LIN {X 0,Y 396.421,Z 620.372,A -85,B 0,C 180,E1 -11060.818,E2 -11060.818} C_VEL
LIN {X 0,Y 396.005,Z 626.08,A -85,B 0,C 180,E1 -11062.862,E2 -11062.862} C_VEL
LIN {X 0,Y 395.858,Z 630.229,A -85,B 0,C 180,E1 -11064.906,E2 -11064.906} C_VEL
LIN {X 0,Y 395.697,Z 632.948,A -85,B 0,C 180,E1 -11066.944,E2 -11066.944} C_VEL
LIN {X 0,Y 395.755,Z 634.313,A -85,B 0,C 180,E1 -11068.981,E2 -11068.981} C_VEL
LIN {X 0,Y 395.755,Z 634.351,A -85,B 0,C 180,E1 -11071.016,E2 -11071.016} C_VEL
LIN {X 0,Y 395.696,Z 633.059,A -85,B 0,C 180,E1 -11073.053,E2 -11073.053} C_VEL
LIN {X 0,Y 395.856,Z 630.406,A -85,B 0,C 180,E1 -11075.091,E2 -11075.091} C_VEL
LIN {X 0,Y 396.003,Z 626.321,A -85,B 0,C 180,E1 -11077.135,E2 -11077.135} C_VEL
LIN {X 0,Y 396.407,Z 620.682,A -85,B 0,C 180,E1 -11079.18,E2 -11079.18} C_VEL
LIN {X 0,Y 396.918,Z 614.321,A -85,B 0,C 180,E1 -11080.971,E2 -11080.971} C_VEL
LIN {X 0,Y 397.802,Z 606.411,A -85,B 0,C 180,E1 -11082.757,E2 -11082.757} C_VEL
LIN {X 0,Y 398.55,Z 598.138,A -85,B 0,C 180,E1 -11084.291,E2 -11084.291} C_VEL
LIN {X 0,Y 399.604,Z 588.172,A -85,B 0,C 180,E1 -11085.818,E2 -11085.818} C_VEL
LIN {X 0,Y 400.764,Z 577.081,A -85,B 0,C 180,E1 -11087.212,E2 -11087.212} C_VEL
LIN {X 0,Y 401.87,Z 566.044,A -85,B 0,C 180,E1 -11088.347,E2 -11088.347} C_VEL
LIN {X 0,Y 402.968,Z 554.065,A -85,B 0,C 180,E1 -11089.35,E2 -11089.35} C_VEL
LIN {X 0,Y 404.005,Z 540.311,A -85,B 0,C 180,E1 -11090.255,E2 -11090.255} C_VEL
LIN {X 0,Y 404.838,Z 526.291,A -85,B 0,C 180,E1 -11090.946,E2 -11090.946} C_VEL
LIN {X 0,Y 405.521,Z 512.757,A -85,B 0,C 180,E1 -11091.408,E2 -11091.408} C_VEL
LIN {X 0,Y 405.97,Z 492.817,A -85,B 0,C 180,E1 -11091.816,E2 -11091.816} C_VEL
LIN {X 0,Y 407.438,Z 401.297,A -85,B 0,C 180,E1 -11093.445,E2 -11093.445} C_VEL
LIN {X 0,Y 402.179,Z 375.662,A -85,B 0,C 180,E1 -11094.261,E2 -11094.261} C_VEL
LIN {X 0,Y 401.525,Z 372.237,A -85,B 0,C 180,E1 -11094.402,E2 -11094.402} C_VEL
LIN {X 0,Y 401.284,Z 368.64,A -85,B 0,C 180,E1 -11095.131,E2 -11095.131} C_VEL
LIN {X 0,Y 398.971,Z 357.321,A -85,B 0,C 180,E1 -11097.727,E2 -11097.727} C_VEL
LIN {X 0,Y 397.187,Z 349.822,A -85,B 0,C 180,E1 -11099.551,E2 -11099.551} C_VEL
LIN {X 0,Y 397.111,Z 349.638,A -85,B 0,C 180,E1 -11103.271,E2 -11103.271} C_VEL
LIN {X 0,Y 397.105,Z 349.636,A -85,B 0,C 180,E1 -11105.733,E2 -11105.733} C_VEL
LIN {X 0,Y 397.111,Z 349.632,A -85,B 0,C 180,E1 -11109.575,E2 -11109.575} C_VEL
LIN {X 0,Y 397.154,Z 349.64,A -85,B 0,C 180,E1 -11112.254,E2 -11112.254} C_VEL
LIN {X 0,Y 397.145,Z 349.618,A -85,B 0,C 180,E1 -11115.058,E2 -11115.058} C_VEL
LIN {X 0,Y 397.149,Z 349.642,A -85,B 0,C 180,E1 -11118.005,E2 -11118.005} C_VEL
LIN {X 0,Y 397.102,Z 349.617,A -85,B 0,C 180,E1 -11121.725,E2 -11121.725} C_VEL
LIN {X 0,Y 397.117,Z 349.642,A -85,B 0,C 180,E1 -11125.506,E2 -11125.506} C_VEL
LIN {X 0,Y 397.076,Z 349.628,A -85,B 0,C 180,E1 -11129.117,E2 -11129.117} C_VEL
LIN {X 0,Y 397.185,Z 349.612,A -85,B 0,C 180,E1 -11132.609,E2 -11132.609} C_VEL
LIN {X 0,Y 397.124,Z 349.642,A -85,B 0,C 180,E1 -11135.981,E2 -11135.981} C_VEL
LIN {X 0,Y 397.128,Z 349.636,A -85,B 0,C 180,E1 -11139.704,E2 -11139.704} C_VEL
LIN {X 0,Y 397.171,Z 349.634,A -85,B 0,C 180,E1 -11142.844,E2 -11142.844} C_VEL
LIN {X 0,Y 397.215,Z 349.626,A -85,B 0,C 180,E1 -11146.678,E2 -11146.678} C_VEL
LIN {X 0,Y 397.219,Z 349.615,A -85,B 0,C 180,E1 -11149.809,E2 -11149.809} C_VEL
LIN {X 0,Y 397.354,Z 349.611,A -85,B 0,C 180,E1 -11152.888,E2 -11152.888} C_VEL
LIN {X 0,Y 397.248,Z 349.625,A -85,B 0,C 180,E1 -11154.925,E2 -11154.925} C_VEL
LIN {X 0,Y 397.442,Z 349.595,A -85,B 0,C 180,E1 -11157.973,E2 -11157.973} C_VEL
LIN {X 0,Y 397.574,Z 349.584,A -85,B 0,C 180,E1 -11160,E2 -11160} C_VEL
LIN {X 0,Y 397.374,Z 349.599,A -85,B 0,C 180,E1 -11163.041,E2 -11163.041} C_VEL
LIN {X 0,Y 397.353,Z 349.611,A -85,B 0,C 180,E1 -11167.112,E2 -11167.112} C_VEL
LIN {X 0,Y 397.219,Z 349.615,A -85,B 0,C 180,E1 -11170.191,E2 -11170.191} C_VEL
LIN {X 0,Y 397.215,Z 349.625,A -85,B 0,C 180,E1 -11173.321,E2 -11173.321} C_VEL
LIN {X 0,Y 397.171,Z 349.633,A -85,B 0,C 180,E1 -11177.156,E2 -11177.156} C_VEL
LIN {X 0,Y 397.104,Z 349.634,A -85,B 0,C 180,E1 -11180.73,E2 -11180.73} C_VEL
LIN {X 0,Y 397.124,Z 349.641,A -85,B 0,C 180,E1 -11184.019,E2 -11184.019} C_VEL
LIN {X 0,Y 397.184,Z 349.612,A -85,B 0,C 180,E1 -11187.391,E2 -11187.391} C_VEL
LIN {X 0,Y 397.069,Z 349.628,A -85,B 0,C 180,E1 -11190.883,E2 -11190.883} C_VEL
LIN {X 0,Y 397.117,Z 349.642,A -85,B 0,C 180,E1 -11194.494,E2 -11194.494} C_VEL
LIN {X 0,Y 397.101,Z 349.616,A -85,B 0,C 180,E1 -11198.275,E2 -11198.275} C_VEL
LIN {X 0,Y 397.149,Z 349.642,A -85,B 0,C 180,E1 -11201.995,E2 -11201.995} C_VEL
LIN {X 0,Y 397.144,Z 349.618,A -85,B 0,C 180,E1 -11205.061,E2 -11205.061} C_VEL
LIN {X 0,Y 397.15,Z 349.641,A -85,B 0,C 180,E1 -11208.008,E2 -11208.008} C_VEL
LIN {X 0,Y 397.104,Z 349.643,A -85,B 0,C 180,E1 -11211.727,E2 -11211.727} C_VEL
LIN {X 0,Y 397.121,Z 349.643,A -85,B 0,C 180,E1 -11215.508,E2 -11215.508} C_VEL
LIN {X 0,Y 397.084,Z 349.641,A -85,B 0,C 180,E1 -11219.12,E2 -11219.12} C_VEL
LIN {X 0,Y 397.147,Z 349.731,A -85,B 0,C 180,E1 -11220.445,E2 -11220.445} C_VEL
LIN {X 0,Y 399.635,Z 360.386,A -85,B 0,C 180,E1 -11223.033,E2 -11223.033} C_VEL
LIN {X 0,Y 401.501,Z 369.735,A -85,B 0,C 180,E1 -11225.161,E2 -11225.161} C_VEL
LIN {X 0,Y 401.565,Z 372.2,A -85,B 0,C 180,E1 -11225.642,E2 -11225.642} C_VEL
LIN {X 0,Y 405.138,Z 389.382,A -85,B 0,C 180,E1 -11226.233,E2 -11226.233} C_VEL
LIN {X 0,Y 407.399,Z 401.324,A -85,B 0,C 180,E1 -11226.598,E2 -11226.598} C_VEL
LIN {X 0,Y 405.977,Z 492.194,A -85,B 0,C 180,E1 -11228.217,E2 -11228.217} C_VEL
LIN {X 0,Y 405.512,Z 512.358,A -85,B 0,C 180,E1 -11228.625,E2 -11228.625} C_VEL
LIN {X 0,Y 404.83,Z 526.784,A -85,B 0,C 180,E1 -11229.12,E2 -11229.12} C_VEL
LIN {X 0,Y 404.089,Z 539.32,A -85,B 0,C 180,E1 -11229.736,E2 -11229.736} C_VEL
LIN {X 0,Y 403.167,Z 552.336,A -85,B 0,C 180,E1 -11230.574,E2 -11230.574} C_VEL
LIN {X 0,Y 402.127,Z 564.159,A -85,B 0,C 180,E1 -11231.534,E2 -11231.534} C_VEL
LIN {X 0,Y 400.922,Z 575.526,A -85,B 0,C 180,E1 -11232.664,E2 -11232.664} C_VEL
LIN {X 0,Y 399.832,Z 585.975,A -85,B 0,C 180,E1 -11233.93,E2 -11233.93} C_VEL
LIN {X 0,Y 398.709,Z 596.365,A -85,B 0,C 180,E1 -11235.454,E2 -11235.454} C_VEL
LIN {X 0,Y 397.963,Z 604.935,A -85,B 0,C 180,E1 -11236.989,E2 -11236.989} C_VEL
LIN {X 0,Y 397.035,Z 613.139,A -85,B 0,C 180,E1 -11238.773,E2 -11238.773} C_VEL
LIN {X 0,Y 396.57,Z 618.879,A -85,B 0,C 180,E1 -11240.309,E2 -11240.309} C_VEL
LIN {X 0,Y 396.17,Z 623.58,A -85,B 0,C 180,E1 -11241.842,E2 -11241.842} C_VEL
LIN {X 0,Y 395.948,Z 628.456,A -85,B 0,C 180,E1 -11243.888,E2 -11243.888} C_VEL
LIN {X 0,Y 395.772,Z 631.842,A -85,B 0,C 180,E1 -11245.928,E2 -11245.928} C_VEL
LIN {X 0,Y 395.719,Z 633.84,A -85,B 0,C 180,E1 -11247.966,E2 -11247.966} C_VEL
LIN {X 0,Y 395.725,Z 634.5,A -85,B 0,C 180,E1 -11250.001,E2 -11250.001} C_VEL
LIN {X 0,Y 395.719,Z 633.832,A -85,B 0,C 180,E1 -11252.037,E2 -11252.037} C_VEL
LIN {X 0,Y 395.772,Z 631.825,A -85,B 0,C 180,E1 -11254.074,E2 -11254.074} C_VEL
LIN {X 0,Y 395.91,Z 628.434,A -85,B 0,C 180,E1 -11256.115,E2 -11256.115} C_VEL
LIN {X 0,Y 396.173,Z 623.556,A -85,B 0,C 180,E1 -11258.16,E2 -11258.16} C_VEL
LIN {X 0,Y 396.725,Z 617.037,A -85,B 0,C 180,E1 -11260.205,E2 -11260.205} C_VEL
LIN {X 0,Y 397.444,Z 609.781,A -85,B 0,C 180,E1 -11261.993,E2 -11261.993} C_VEL
LIN {X 0,Y 398.133,Z 602.2,A -85,B 0,C 180,E1 -11263.523,E2 -11263.523} C_VEL
LIN {X 0,Y 399.052,Z 593.048,A -85,B 0,C 180,E1 -11265.058,E2 -11265.058} C_VEL
LIN {X 0,Y 400.235,Z 581.976,A -85,B 0,C 180,E1 -11266.581,E2 -11266.581} C_VEL
LIN {X 0,Y 401.442,Z 570.666,A -85,B 0,C 180,E1 -11267.842,E2 -11267.842} C_VEL
LIN {X 0,Y 402.603,Z 558.152,A -85,B 0,C 180,E1 -11268.974,E2 -11268.974} C_VEL
LIN {X 0,Y 403.664,Z 544.973,A -85,B 0,C 180,E1 -11269.92,E2 -11269.92} C_VEL
LIN {X 0,Y 404.508,Z 531.447,A -85,B 0,C 180,E1 -11270.667,E2 -11270.667} C_VEL
LIN {X 0,Y 405.258,Z 517.305,A -85,B 0,C 180,E1 -11271.225,E2 -11271.225} C_VEL
LIN {X 0,Y 405.747,Z 502.321,A -85,B 0,C 180,E1 -11271.598,E2 -11271.598} C_VEL
LIN {X 0,Y 407.395,Z 404.163,A -85,B 0,C 180,E1 -11273.34,E2 -11273.34} C_VEL
LIN {X 0,Y 407.089,Z 399.782,A -85,B 0,C 180,E1 -11273.441,E2 -11273.441} C_VEL
LIN {X 0,Y 401.913,Z 374.308,A -85,B 0,C 180,E1 -11274.249,E2 -11274.249} C_VEL
LIN {X 0,Y 401.579,Z 371.957,A -85,B 0,C 180,E1 -11274.385,E2 -11274.385} C_VEL
LIN {X 0,Y 400.995,Z 367.058,A -85,B 0,C 180,E1 -11275.43,E2 -11275.43} C_VEL
LIN {X 0,Y 398.157,Z 353.978,A -85,B 0,C 180,E1 -11278.464,E2 -11278.464} C_VEL
LIN {X 0,Y 397.143,Z 349.691,A -85,B 0,C 180,E1 -11279.558,E2 -11279.558} C_VEL
LIN {X 0,Y 397.119,Z 349.642,A -85,B 0,C 180,E1 -11283.274,E2 -11283.274} C_VEL
LIN {X 0,Y 397.114,Z 349.644,A -85,B 0,C 180,E1 -11285.735,E2 -11285.735} C_VEL
LIN {X 0,Y 397.119,Z 349.642,A -85,B 0,C 180,E1 -11289.578,E2 -11289.578} C_VEL
LIN {X 0,Y 397.107,Z 349.644,A -85,B 0,C 180,E1 -11293.48,E2 -11293.48} C_VEL
LIN {X 0,Y 397.107,Z 349.644,A -85,B 0,C 180,E1 -11296.522,E2 -11296.522} C_VEL
LIN {X 0,Y 397.118,Z 349.645,A -85,B 0,C 180,E1 -11300.423,E2 -11300.423} C_VEL
LIN {X 0,Y 397.113,Z 349.647,A -85,B 0,C 180,E1 -11304.266,E2 -11304.266} C_VEL
LIN {X 0,Y 397.134,Z 349.794,A -85,B 0,C 180,E1 -11305.888,E2 -11305.888} C_VEL
LIN {X 0,Y 400.499,Z 359.333,A -85,B 0,C 180,E1 -11308.235,E2 -11308.235} C_VEL
LIN {X 0,Y 403.186,Z 368.452,A -85,B 0,C 180,E1 -11310.213,E2 -11310.213} C_VEL
LIN {X 0,Y 404.815,Z 376.269,A -85,B 0,C 180,E1 -11311.765,E2 -11311.765} C_VEL
LIN {X 0,Y 404.96,Z 379.108,A -85,B 0,C 180,E1 -11312.265,E2 -11312.265} C_VEL
LIN {X 0,Y 403.241,Z 401.255,A -85,B 0,C 180,E1 -11315.822,E2 -11315.822} C_VEL
LIN {X 0,Y 401.955,Z 420.536,A -85,B 0,C 180,E1 -11318.845,E2 -11318.845} C_VEL
LIN {X 0,Y 404.754,Z 435.53,A -85,B 0,C 180,E1 -11319.532,E2 -11319.532} C_VEL
LIN {X 0,Y 405.919,Z 445.255,A -85,B 0,C 180,E1 -11319.902,E2 -11319.902} C_VEL
LIN {X 0,Y 403.283,Z 522.514,A -85,B 0,C 180,E1 -11321.817,E2 -11321.817} C_VEL
LIN {X 0,Y 402.775,Z 537.366,A -85,B 0,C 180,E1 -11322.253,E2 -11322.253} C_VEL
LIN {X 0,Y 402.105,Z 549.391,A -85,B 0,C 180,E1 -11322.781,E2 -11322.781} C_VEL
LIN {X 0,Y 401.225,Z 562.751,A -85,B 0,C 180,E1 -11323.594,E2 -11323.594} C_VEL
LIN {X 0,Y 400.405,Z 573.966,A -85,B 0,C 180,E1 -11324.474,E2 -11324.474} C_VEL
LIN {X 0,Y 399.44,Z 584.575,A -85,B 0,C 180,E1 -11325.514,E2 -11325.514} C_VEL
LIN {X 0,Y 398.635,Z 594.744,A -85,B 0,C 180,E1 -11326.751,E2 -11326.751} C_VEL
LIN {X 0,Y 397.863,Z 603.355,A -85,B 0,C 180,E1 -11328.021,E2 -11328.021} C_VEL
LIN {X 0,Y 397.204,Z 611.715,A -85,B 0,C 180,E1 -11329.551,E2 -11329.551} C_VEL
LIN {X 0,Y 396.628,Z 618.463,A -85,B 0,C 180,E1 -11331.081,E2 -11331.081} C_VEL
LIN {X 0,Y 396.148,Z 624.608,A -85,B 0,C 180,E1 -11332.866,E2 -11332.866} C_VEL
LIN {X 0,Y 395.985,Z 628.555,A -85,B 0,C 180,E1 -11334.398,E2 -11334.398} C_VEL
LIN {X 0,Y 395.796,Z 631.423,A -85,B 0,C 180,E1 -11335.927,E2 -11335.927} C_VEL
LIN {X 0,Y 395.717,Z 632.768,A -85,B 0,C 180,E1 -11336.946,E2 -11336.946} C_VEL
LIN {X 0,Y 395.742,Z 633.695,A -85,B 0,C 180,E1 -11337.965,E2 -11337.965} C_VEL
LIN {X 0,Y 395.759,Z 634.149,A -85,B 0,C 180,E1 -11338.983,E2 -11338.983} C_VEL
LIN {X 0,Y 395.728,Z 634.175,A -85,B 0,C 180,E1 -11340,E2 -11340} C_VEL
LIN {X 0,Y 395.758,Z 633.789,A -85,B 0,C 180,E1 -11341.018,E2 -11341.018} C_VEL
LIN {X 0,Y 395.724,Z 632.943,A -85,B 0,C 180,E1 -11342.036,E2 -11342.036} C_VEL
LIN {X 0,Y 395.703,Z 631.648,A -85,B 0,C 180,E1 -11343.054,E2 -11343.054} C_VEL
LIN {X 0,Y 395.861,Z 628.869,A -85,B 0,C 180,E1 -11344.582,E2 -11344.582} C_VEL
LIN {X 0,Y 395.949,Z 624.513,A -85,B 0,C 180,E1 -11346.28,E2 -11346.28} C_VEL
LIN {X 0,Y 396.19,Z 618.946,A -85,B 0,C 180,E1 -11347.902,E2 -11347.902} C_VEL
LIN {X 0,Y 396.512,Z 612.231,A -85,B 0,C 180,E1 -11349.436,E2 -11349.436} C_VEL
LIN {X 0,Y 396.979,Z 603.876,A -85,B 0,C 180,E1 -11350.971,E2 -11350.971} C_VEL
LIN {X 0,Y 397.57,Z 595.271,A -85,B 0,C 180,E1 -11352.247,E2 -11352.247} C_VEL
LIN {X 0,Y 398.246,Z 585.343,A -85,B 0,C 180,E1 -11353.453,E2 -11353.453} C_VEL
LIN {X 0,Y 398.827,Z 574.328,A -85,B 0,C 180,E1 -11354.543,E2 -11354.543} C_VEL
LIN {X 0,Y 399.433,Z 562.909,A -85,B 0,C 180,E1 -11355.434,E2 -11355.434} C_VEL
LIN {X 0,Y 400.096,Z 550.33,A -85,B 0,C 180,E1 -11356.192,E2 -11356.192} C_VEL
LIN {X 0,Y 400.582,Z 537.225,A -85,B 0,C 180,E1 -11356.762,E2 -11356.762} C_VEL
LIN {X 0,Y 400.934,Z 523.753,A -85,B 0,C 180,E1 -11357.14,E2 -11357.14} C_VEL
LIN {X 0,Y 402.464,Z 443.323,A -85,B 0,C 180,E1 -11358.914,E2 -11358.914} C_VEL
LIN {X 0,Y 399.497,Z 420.826,A -85,B 0,C 180,E1 -11359.56,E2 -11359.56} C_VEL
LIN {X 0,Y 400.434,Z 402.169,A -85,B 0,C 180,E1 -11362.441,E2 -11362.441} C_VEL
LIN {X 0,Y 401.562,Z 381.596,A -85,B 0,C 180,E1 -11365.669,E2 -11365.669} C_VEL
LIN {X 0,Y 402.022,Z 372.95,A -85,B 0,C 180,E1 -11367.034,E2 -11367.034} C_VEL
LIN {X 0,Y 401.183,Z 367.577,A -85,B 0,C 180,E1 -11367.944,E2 -11367.944} C_VEL
LIN {X 0,Y 397.131,Z 349.787,A -85,B 0,C 180,E1 -11371.1,E2 -11371.1} C_VEL
LIN {X 0,Y 397.131,Z 349.644,A -85,B 0,C 180,E1 -11374.493,E2 -11374.493} C_VEL
LIN {X 0,Y 397.105,Z 349.647,A -85,B 0,C 180,E1 -11378.275,E2 -11378.275} C_VEL
LIN {X 0,Y 397.094,Z 349.645,A -85,B 0,C 180,E1 -11380.908,E2 -11380.908} C_VEL
LIN {X 0,Y 397.106,Z 349.634,A -85,B 0,C 180,E1 -11383.648,E2 -11383.648} C_VEL
LIN {X 0,Y 397.108,Z 349.638,A -85,B 0,C 180,E1 -11386.52,E2 -11386.52} C_VEL
LIN {X 0,Y 397.12,Z 349.63,A -85,B 0,C 180,E1 -11390.422,E2 -11390.422} C_VEL
LIN {X 0,Y 397.115,Z 349.634,A -85,B 0,C 180,E1 -11394.265,E2 -11394.265} C_VEL
LIN {X 0,Y 397.12,Z 349.638,A -85,B 0,C 180,E1 -11396.726,E2 -11396.726} C_VEL
LIN {X 0,Y 397.186,Z 349.732,A -85,B 0,C 180,E1 -11400.518,E2 -11400.518} C_VEL
LIN {X 0,Y 399.829,Z 361.267,A -85,B 0,C 180,E1 -11403.293,E2 -11403.293} C_VEL
LIN {X 0,Y 401.589,Z 371.098,A -85,B 0,C 180,E1 -11405.509,E2 -11405.509} C_VEL
LIN {X 0,Y 401.574,Z 372.504,A -85,B 0,C 180,E1 -11405.723,E2 -11405.723} C_VEL
LIN {X 0,Y 406.969,Z 399.053,A -85,B 0,C 180,E1 -11406.583,E2 -11406.583} C_VEL
LIN {X 0,Y 407.413,Z 402.849,A -85,B 0,C 180,E1 -11406.682,E2 -11406.682} C_VEL
LIN {X 0,Y 405.619,Z 509.285,A -85,B 0,C 180,E1 -11408.595,E2 -11408.595} C_VEL
LIN {X 0,Y 404.928,Z 523.987,A -85,B 0,C 180,E1 -11409.057,E2 -11409.057} C_VEL
LIN {X 0,Y 404.229,Z 536.848,A -85,B 0,C 180,E1 -11409.651,E2 -11409.651} C_VEL
LIN {X 0,Y 403.31,Z 549.904,A -85,B 0,C 180,E1 -11410.452,E2 -11410.452} C_VEL
LIN {X 0,Y 403.06,Z 552.889,A -85,B 0,C 180,E1 -11410.664,E2 -11410.664} C_VEL
LIN {X 0,Y 401.916,Z 558.108,A -85,B 0,C 180,E1 -11411.029,E2 -11411.029} C_VEL
LIN {X 0,Y 398.336,Z 566.424,A -85,B 0,C 180,E1 -11411.619,E2 -11411.619} C_VEL
LIN {X 0,Y 394.805,Z 574.368,A -85,B 0,C 180,E1 -11412.304,E2 -11412.304} C_VEL
LIN {X 0,Y 393.743,Z 578.997,A -85,B 0,C 180,E1 -11412.81,E2 -11412.81} C_VEL
LIN {X 0,Y 392.61,Z 589.273,A -85,B 0,C 180,E1 -11414.157,E2 -11414.157} C_VEL
LIN {X 0,Y 391.426,Z 599.739,A -85,B 0,C 180,E1 -11415.828,E2 -11415.828} C_VEL
LIN {X 0,Y 390.606,Z 608.4,A -85,B 0,C 180,E1 -11417.53,E2 -11417.53} C_VEL
LIN {X 0,Y 389.852,Z 614.941,A -85,B 0,C 180,E1 -11419.088,E2 -11419.088} C_VEL
LIN {X 0,Y 389.387,Z 620.373,A -85,B 0,C 180,E1 -11420.65,E2 -11420.65} C_VEL
LIN {X 0,Y 388.934,Z 626.082,A -85,B 0,C 180,E1 -11422.732,E2 -11422.732} C_VEL
LIN {X 0,Y 388.778,Z 630.23,A -85,B 0,C 180,E1 -11424.813,E2 -11424.813} C_VEL
LIN {X 0,Y 388.608,Z 632.948,A -85,B 0,C 180,E1 -11426.889,E2 -11426.889} C_VEL
LIN {X 0,Y 388.654,Z 634.313,A -85,B 0,C 180,E1 -11428.963,E2 -11428.963} C_VEL
LIN {X 0,Y 388.654,Z 634.35,A -85,B 0,C 180,E1 -11431.035,E2 -11431.035} C_VEL
LIN {X 0,Y 388.606,Z 633.059,A -85,B 0,C 180,E1 -11433.109,E2 -11433.109} C_VEL
LIN {X 0,Y 388.757,Z 630.406,A -85,B 0,C 180,E1 -11435.185,E2 -11435.185} C_VEL
LIN {X 0,Y 388.931,Z 626.32,A -85,B 0,C 180,E1 -11437.265,E2 -11437.265} C_VEL
LIN {X 0,Y 389.372,Z 620.681,A -85,B 0,C 180,E1 -11439.347,E2 -11439.347} C_VEL
LIN {X 0,Y 389.917,Z 614.319,A -85,B 0,C 180,E1 -11441.171,E2 -11441.171} C_VEL
LIN {X 0,Y 390.847,Z 606.409,A -85,B 0,C 180,E1 -11442.988,E2 -11442.988} C_VEL
LIN {X 0,Y 391.641,Z 598.135,A -85,B 0,C 180,E1 -11444.549,E2 -11444.549} C_VEL
LIN {X 0,Y 392.755,Z 588.169,A -85,B 0,C 180,E1 -11446.101,E2 -11446.101} C_VEL
LIN {X 0,Y 393.97,Z 577.077,A -85,B 0,C 180,E1 -11447.518,E2 -11447.518} C_VEL
LIN {X 0,Y 395.113,Z 566.04,A -85,B 0,C 180,E1 -11448.672,E2 -11448.672} C_VEL
LIN {X 0,Y 396.275,Z 554.059,A -85,B 0,C 180,E1 -11449.691,E2 -11449.691} C_VEL
LIN {X 0,Y 397.343,Z 540.457,A -85,B 0,C 180,E1 -11450.601,E2 -11450.601} C_VEL
LIN {X 0,Y 398.185,Z 527.042,A -85,B 0,C 180,E1 -11451.279,E2 -11451.279} C_VEL
LIN {X 0,Y 398.943,Z 512.741,A -85,B 0,C 180,E1 -11451.779,E2 -11451.779} C_VEL
LIN {X 0,Y 399.409,Z 492.791,A -85,B 0,C 180,E1 -11452.194,E2 -11452.194} C_VEL
LIN {X 0,Y 400.871,Z 402.203,A -85,B 0,C 180,E1 -11453.835,E2 -11453.835} C_VEL
LIN {X 0,Y 395.647,Z 376.514,A -85,B 0,C 180,E1 -11454.671,E2 -11454.671} C_VEL
LIN {X 0,Y 394.684,Z 372.069,A -85,B 0,C 180,E1 -11454.871,E2 -11454.871} C_VEL
LIN {X 0,Y 392.774,Z 362.1,A -85,B 0,C 180,E1 -11457.145,E2 -11457.145} C_VEL
LIN {X 0,Y 390.119,Z 350.792,A -85,B 0,C 180,E1 -11459.91,E2 -11459.91} C_VEL
LIN {X 0,Y 390.042,Z 350.504,A -85,B 0,C 180,E1 -11460.298,E2 -11460.298} C_VEL
LIN {X 0,Y 390.08,Z 350.52,A -85,B 0,C 180,E1 -11463.952,E2 -11463.952} C_VEL
LIN {X 0,Y 390.043,Z 350.525,A -85,B 0,C 180,E1 -11467.55,E2 -11467.55} C_VEL
LIN {X 0,Y 390.077,Z 350.512,A -85,B 0,C 180,E1 -11470.825,E2 -11470.825} C_VEL
LIN {X 0,Y 390.123,Z 350.502,A -85,B 0,C 180,E1 -11473.896,E2 -11473.896} C_VEL
LIN {X 0,Y 390.111,Z 350.508,A -85,B 0,C 180,E1 -11476.797,E2 -11476.797} C_VEL
LIN {X 0,Y 390.071,Z 350.518,A -85,B 0,C 180,E1 -11479.562,E2 -11479.562} C_VEL
LIN {X 0,Y 390.039,Z 350.494,A -85,B 0,C 180,E1 -11482.447,E2 -11482.447} C_VEL
LIN {X 0,Y 390.075,Z 350.522,A -85,B 0,C 180,E1 -11486.046,E2 -11486.046} C_VEL
LIN {X 0,Y 390.043,Z 350.491,A -85,B 0,C 180,E1 -11489.867,E2 -11489.867} C_VEL
LIN {X 0,Y 390.104,Z 350.497,A -85,B 0,C 180,E1 -11493.231,E2 -11493.231} C_VEL
LIN {X 0,Y 390.097,Z 350.516,A -85,B 0,C 180,E1 -11496.749,E2 -11496.749} C_VEL
LIN {X 0,Y 390.094,Z 350.514,A -85,B 0,C 180,E1 -11499.982,E2 -11499.982} C_VEL
LIN {X 0,Y 390.127,Z 350.506,A -85,B 0,C 180,E1 -11503.248,E2 -11503.248} C_VEL
LIN {X 0,Y 390.184,Z 350.501,A -85,B 0,C 180,E1 -11506.561,E2 -11506.561} C_VEL
LIN {X 0,Y 390.169,Z 350.495,A -85,B 0,C 180,E1 -11509.623,E2 -11509.623} C_VEL
LIN {X 0,Y 390.308,Z 350.487,A -85,B 0,C 180,E1 -11512.759,E2 -11512.759} C_VEL
LIN {X 0,Y 390.22,Z 350.501,A -85,B 0,C 180,E1 -11514.833,E2 -11514.833} C_VEL
LIN {X 0,Y 390.411,Z 350.471,A -85,B 0,C 180,E1 -11517.937,E2 -11517.937} C_VEL
LIN {X 0,Y 390.543,Z 350.46,A -85,B 0,C 180,E1 -11520,E2 -11520} C_VEL
LIN {X 0,Y 390.308,Z 350.478,A -85,B 0,C 180,E1 -11523.096,E2 -11523.096} C_VEL
LIN {X 0,Y 390.321,Z 350.486,A -85,B 0,C 180,E1 -11526.202,E2 -11526.202} C_VEL
LIN {X 0,Y 390.304,Z 350.486,A -85,B 0,C 180,E1 -11528.282,E2 -11528.282} C_VEL
LIN {X 0,Y 390.168,Z 350.506,A -85,B 0,C 180,E1 -11532.483,E2 -11532.483} C_VEL
LIN {X 0,Y 390.129,Z 350.496,A -85,B 0,C 180,E1 -11535.677,E2 -11535.677} C_VEL
LIN {X 0,Y 390.095,Z 350.515,A -85,B 0,C 180,E1 -11538.923,E2 -11538.923} C_VEL
LIN {X 0,Y 390.03,Z 350.516,A -85,B 0,C 180,E1 -11542.235,E2 -11542.235} C_VEL
LIN {X 0,Y 390.109,Z 350.51,A -85,B 0,C 180,E1 -11545.744,E2 -11545.744} C_VEL
LIN {X 0,Y 390.047,Z 350.482,A -85,B 0,C 180,E1 -11549.11,E2 -11549.11} C_VEL
LIN {X 0,Y 390.033,Z 350.526,A -85,B 0,C 180,E1 -11552.722,E2 -11552.722} C_VEL
LIN {X 0,Y 390.048,Z 350.512,A -85,B 0,C 180,E1 -11555.827,E2 -11555.827} C_VEL
LIN {X 0,Y 390.066,Z 350.505,A -85,B 0,C 180,E1 -11559.22,E2 -11559.22} C_VEL
LIN {X 0,Y 390.114,Z 350.513,A -85,B 0,C 180,E1 -11562.388,E2 -11562.388} C_VEL
LIN {X 0,Y 390.112,Z 350.495,A -85,B 0,C 180,E1 -11565.366,E2 -11565.366} C_VEL
LIN {X 0,Y 390.099,Z 350.517,A -85,B 0,C 180,E1 -11568.198,E2 -11568.198} C_VEL
LIN {X 0,Y 390.089,Z 350.509,A -85,B 0,C 180,E1 -11570.91,E2 -11570.91} C_VEL
LIN {X 0,Y 390.08,Z 350.513,A -85,B 0,C 180,E1 -11574.795,E2 -11574.795} C_VEL
LIN {X 0,Y 390.045,Z 350.527,A -85,B 0,C 180,E1 -11578.499,E2 -11578.499} C_VEL
LIN {X 0,Y 390.092,Z 350.67,A -85,B 0,C 180,E1 -11580.088,E2 -11580.088} C_VEL
LIN {X 0,Y 392.741,Z 361.896,A -85,B 0,C 180,E1 -11582.853,E2 -11582.853} C_VEL
LIN {X 0,Y 394.744,Z 372.239,A -85,B 0,C 180,E1 -11585.197,E2 -11585.197} C_VEL
LIN {X 0,Y 397.117,Z 383.368,A -85,B 0,C 180,E1 -11585.605,E2 -11585.605} C_VEL
LIN {X 0,Y 400.904,Z 402.788,A -85,B 0,C 180,E1 -11586.223,E2 -11586.223} C_VEL
LIN {X 0,Y 399.133,Z 505.902,A -85,B 0,C 180,E1 -11588.096,E2 -11588.096} C_VEL
LIN {X 0,Y 398.545,Z 520.359,A -85,B 0,C 180,E1 -11588.504,E2 -11588.504} C_VEL
LIN {X 0,Y 397.703,Z 534.258,A -85,B 0,C 180,E1 -11589.101,E2 -11589.101} C_VEL
LIN {X 0,Y 396.857,Z 547.06,A -85,B 0,C 180,E1 -11589.857,E2 -11589.857} C_VEL
LIN {X 0,Y 395.768,Z 559.865,A -85,B 0,C 180,E1 -11590.823,E2 -11590.823} C_VEL
LIN {X 0,Y 394.534,Z 572.01,A -85,B 0,C 180,E1 -11591.972,E2 -11591.972} C_VEL
LIN {X 0,Y 393.448,Z 582.061,A -85,B 0,C 180,E1 -11593.128,E2 -11593.128} C_VEL
LIN {X 0,Y 392.184,Z 593.114,A -85,B 0,C 180,E1 -11594.675,E2 -11594.675} C_VEL
LIN {X 0,Y 391.149,Z 602.56,A -85,B 0,C 180,E1 -11596.293,E2 -11596.293} C_VEL
LIN {X 0,Y 390.463,Z 609.826,A -85,B 0,C 180,E1 -11597.792,E2 -11597.792} C_VEL
LIN {X 0,Y 389.701,Z 617.072,A -85,B 0,C 180,E1 -11599.612,E2 -11599.612} C_VEL
LIN {X 0,Y 389.114,Z 623.581,A -85,B 0,C 180,E1 -11601.694,E2 -11601.694} C_VEL
LIN {X 0,Y 388.872,Z 628.457,A -85,B 0,C 180,E1 -11603.776,E2 -11603.776} C_VEL
LIN {X 0,Y 388.698,Z 631.842,A -85,B 0,C 180,E1 -11605.854,E2 -11605.854} C_VEL
LIN {X 0,Y 388.616,Z 633.841,A -85,B 0,C 180,E1 -11607.929,E2 -11607.929} C_VEL
LIN {X 0,Y 388.639,Z 634.5,A -85,B 0,C 180,E1 -11610.001,E2 -11610.001} C_VEL
LIN {X 0,Y 388.617,Z 633.832,A -85,B 0,C 180,E1 -11612.074,E2 -11612.074} C_VEL
LIN {X 0,Y 388.698,Z 631.824,A -85,B 0,C 180,E1 -11614.149,E2 -11614.149} C_VEL
LIN {X 0,Y 388.834,Z 628.433,A -85,B 0,C 180,E1 -11616.227,E2 -11616.227} C_VEL
LIN {X 0,Y 389.116,Z 623.555,A -85,B 0,C 180,E1 -11618.309,E2 -11618.309} C_VEL
LIN {X 0,Y 389.702,Z 617.036,A -85,B 0,C 180,E1 -11620.391,E2 -11620.391} C_VEL
LIN {X 0,Y 390.458,Z 609.78,A -85,B 0,C 180,E1 -11622.211,E2 -11622.211} C_VEL
LIN {X 0,Y 391.286,Z 601.408,A -85,B 0,C 180,E1 -11623.919,E2 -11623.919} C_VEL
LIN {X 0,Y 392.363,Z 591.355,A -85,B 0,C 180,E1 -11625.587,E2 -11625.587} C_VEL
LIN {X 0,Y 393.541,Z 580.907,A -85,B 0,C 180,E1 -11627.005,E2 -11627.005} C_VEL
LIN {X 0,Y 394.798,Z 569.371,A -85,B 0,C 180,E1 -11628.287,E2 -11628.287} C_VEL
LIN {X 0,Y 396.04,Z 556.567,A -85,B 0,C 180,E1 -11629.436,E2 -11629.436} C_VEL
LIN {X 0,Y 397.003,Z 544.862,A -85,B 0,C 180,E1 -11630.276,E2 -11630.276} C_VEL
LIN {X 0,Y 397.883,Z 531.439,A -85,B 0,C 180,E1 -11631.027,E2 -11631.027} C_VEL
LIN {X 0,Y 398.651,Z 517.295,A -85,B 0,C 180,E1 -11631.594,E2 -11631.594} C_VEL
LIN {X 0,Y 399.174,Z 502.302,A -85,B 0,C 180,E1 -11631.972,E2 -11631.972} C_VEL
LIN {X 0,Y 400.895,Z 403.135,A -85,B 0,C 180,E1 -11633.761,E2 -11633.761} C_VEL
LIN {X 0,Y 397.22,Z 383.762,A -85,B 0,C 180,E1 -11634.37,E2 -11634.37} C_VEL
LIN {X 0,Y 394.975,Z 373.194,A -85,B 0,C 180,E1 -11634.736,E2 -11634.736} C_VEL
LIN {X 0,Y 394.615,Z 371.427,A -85,B 0,C 180,E1 -11634.944,E2 -11634.944} C_VEL
LIN {X 0,Y 392.401,Z 360.517,A -85,B 0,C 180,E1 -11637.465,E2 -11637.465} C_VEL
LIN {X 0,Y 390.09,Z 350.626,A -85,B 0,C 180,E1 -11639.914,E2 -11639.914} C_VEL
LIN {X 0,Y 390.089,Z 350.52,A -85,B 0,C 180,E1 -11643.954,E2 -11643.954} C_VEL
LIN {X 0,Y 390.05,Z 350.523,A -85,B 0,C 180,E1 -11647.552,E2 -11647.552} C_VEL
LIN {X 0,Y 390.061,Z 350.521,A -85,B 0,C 180,E1 -11650.822,E2 -11650.822} C_VEL
LIN {X 0,Y 390.059,Z 350.525,A -85,B 0,C 180,E1 -11653.887,E2 -11653.887} C_VEL
LIN {X 0,Y 390.062,Z 350.522,A -85,B 0,C 180,E1 -11656.79,E2 -11656.79} C_VEL
LIN {X 0,Y 390.061,Z 350.522,A -85,B 0,C 180,E1 -11659.561,E2 -11659.561} C_VEL
LIN {X 0,Y 390.048,Z 350.524,A -85,B 0,C 180,E1 -11662.45,E2 -11662.45} C_VEL
LIN {X 0,Y 390.1,Z 350.699,A -85,B 0,C 180,E1 -11664.873,E2 -11664.873} C_VEL
LIN {X 0,Y 393.243,Z 359.102,A -85,B 0,C 180,E1 -11667.139,E2 -11667.139} C_VEL
LIN {X 0,Y 396.584,Z 369.984,A -85,B 0,C 180,E1 -11669.665,E2 -11669.665} C_VEL
LIN {X 0,Y 398.52,Z 379.258,A -85,B 0,C 180,E1 -11671.566,E2 -11671.566} C_VEL
LIN {X 0,Y 398.477,Z 382.61,A -85,B 0,C 180,E1 -11672.154,E2 -11672.154} C_VEL
LIN {X 0,Y 396.647,Z 404.165,A -85,B 0,C 180,E1 -11675.672,E2 -11675.672} C_VEL
LIN {X 0,Y 395.485,Z 420.335,A -85,B 0,C 180,E1 -11678.258,E2 -11678.258} C_VEL
LIN {X 0,Y 398.524,Z 436.321,A -85,B 0,C 180,E1 -11679.047,E2 -11679.047} C_VEL
LIN {X 0,Y 399.634,Z 446.442,A -85,B 0,C 180,E1 -11679.444,E2 -11679.444} C_VEL
LIN {X 0,Y 397.076,Z 514.208,A -85,B 0,C 180,E1 -11681.188,E2 -11681.188} C_VEL
LIN {X 0,Y 396.359,Z 534.94,A -85,B 0,C 180,E1 -11681.756,E2 -11681.756} C_VEL
LIN {X 0,Y 395.656,Z 547.492,A -85,B 0,C 180,E1 -11682.291,E2 -11682.291} C_VEL
LIN {X 0,Y 394.746,Z 560.429,A -85,B 0,C 180,E1 -11683.05,E2 -11683.05} C_VEL
LIN {X 0,Y 393.731,Z 573.51,A -85,B 0,C 180,E1 -11684.071,E2 -11684.071} C_VEL
LIN {X 0,Y 392.665,Z 584.937,A -85,B 0,C 180,E1 -11685.213,E2 -11685.213} C_VEL
LIN {X 0,Y 391.756,Z 595.368,A -85,B 0,C 180,E1 -11686.514,E2 -11686.514} C_VEL
LIN {X 0,Y 390.941,Z 603.842,A -85,B 0,C 180,E1 -11687.806,E2 -11687.806} C_VEL
LIN {X 0,Y 390.232,Z 612.1,A -85,B 0,C 180,E1 -11689.362,E2 -11689.362} C_VEL
LIN {X 0,Y 389.709,Z 617.757,A -85,B 0,C 180,E1 -11690.659,E2 -11690.659} C_VEL
LIN {X 0,Y 389.204,Z 623.275,A -85,B 0,C 180,E1 -11692.217,E2 -11692.217} C_VEL
LIN {X 0,Y 388.926,Z 627.553,A -85,B 0,C 180,E1 -11693.776,E2 -11693.776} C_VEL
LIN {X 0,Y 388.874,Z 629.794,A -85,B 0,C 180,E1 -11694.816,E2 -11694.816} C_VEL
LIN {X 0,Y 388.726,Z 631.535,A -85,B 0,C 180,E1 -11695.853,E2 -11695.853} C_VEL
LIN {X 0,Y 388.627,Z 632.854,A -85,B 0,C 180,E1 -11696.89,E2 -11696.89} C_VEL
LIN {X 0,Y 388.639,Z 633.737,A -85,B 0,C 180,E1 -11697.927,E2 -11697.927} C_VEL
LIN {X 0,Y 388.658,Z 634.149,A -85,B 0,C 180,E1 -11698.964,E2 -11698.964} C_VEL
LIN {X 0,Y 388.642,Z 634.146,A -85,B 0,C 180,E1 -11700,E2 -11700} C_VEL
LIN {X 0,Y 388.657,Z 633.724,A -85,B 0,C 180,E1 -11701.036,E2 -11701.036} C_VEL
LIN {X 0,Y 388.621,Z 632.821,A -85,B 0,C 180,E1 -11702.073,E2 -11702.073} C_VEL
LIN {X 0,Y 388.614,Z 631.49,A -85,B 0,C 180,E1 -11703.11,E2 -11703.11} C_VEL
LIN {X 0,Y 388.771,Z 628.637,A -85,B 0,C 180,E1 -11704.666,E2 -11704.666} C_VEL
LIN {X 0,Y 388.838,Z 624.677,A -85,B 0,C 180,E1 -11706.226,E2 -11706.226} C_VEL
LIN {X 0,Y 389.081,Z 619.513,A -85,B 0,C 180,E1 -11707.786,E2 -11707.786} C_VEL
LIN {X 0,Y 389.403,Z 612.935,A -85,B 0,C 180,E1 -11709.348,E2 -11709.348} C_VEL
LIN {X 0,Y 389.866,Z 604.714,A -85,B 0,C 180,E1 -11710.911,E2 -11710.911} C_VEL
LIN {X 0,Y 390.453,Z 596.321,A -85,B 0,C 180,E1 -11712.21,E2 -11712.21} C_VEL
LIN {X 0,Y 391.1,Z 587.154,A -85,B 0,C 180,E1 -11713.377,E2 -11713.377} C_VEL
LIN {X 0,Y 391.737,Z 575.864,A -85,B 0,C 180,E1 -11714.547,E2 -11714.547} C_VEL
LIN {X 0,Y 392.321,Z 564.938,A -85,B 0,C 180,E1 -11715.454,E2 -11715.454} C_VEL
LIN {X 0,Y 393.057,Z 551.784,A -85,B 0,C 180,E1 -11716.29,E2 -11716.29} C_VEL
LIN {X 0,Y 393.552,Z 538.634,A -85,B 0,C 180,E1 -11716.903,E2 -11716.903} C_VEL
LIN {X 0,Y 393.97,Z 524.713,A -85,B 0,C 180,E1 -11717.319,E2 -11717.319} C_VEL
LIN {X 0,Y 395.525,Z 443.597,A -85,B 0,C 180,E1 -11719.159,E2 -11719.159} C_VEL
LIN {X 0,Y 392.564,Z 420.556,A -85,B 0,C 180,E1 -11719.845,E2 -11719.845} C_VEL
LIN {X 0,Y 393.774,Z 398.004,A -85,B 0,C 180,E1 -11723.398,E2 -11723.398} C_VEL
LIN {X 0,Y 395.133,Z 375.078,A -85,B 0,C 180,E1 -11727.047,E2 -11727.047} C_VEL
LIN {X 0,Y 394.527,Z 370.144,A -85,B 0,C 180,E1 -11727.879,E2 -11727.879} C_VEL
LIN {X 0,Y 390.241,Z 351.464,A -85,B 0,C 180,E1 -11731.194,E2 -11731.194} C_VEL
LIN {X 0,Y 390.093,Z 350.592,A -85,B 0,C 180,E1 -11731.425,E2 -11731.425} C_VEL
LIN {X 0,Y 390.091,Z 350.518,A -85,B 0,C 180,E1 -11735.207,E2 -11735.207} C_VEL
LIN {X 0,Y 390.072,Z 350.519,A -85,B 0,C 180,E1 -11739.217,E2 -11739.217} C_VEL
LIN {X 0,Y 390.048,Z 350.522,A -85,B 0,C 180,E1 -11742.374,E2 -11742.374} C_VEL
LIN {X 0,Y 390.049,Z 350.502,A -85,B 0,C 180,E1 -11745.354,E2 -11745.354} C_VEL
LIN {X 0,Y 390.037,Z 350.526,A -85,B 0,C 180,E1 -11748.186,E2 -11748.186} C_VEL
LIN {X 0,Y 390.097,Z 350.507,A -85,B 0,C 180,E1 -11750.907,E2 -11750.907} C_VEL
LIN {X 0,Y 390.091,Z 350.511,A -85,B 0,C 180,E1 -11754.793,E2 -11754.793} C_VEL
LIN {X 0,Y 390.037,Z 350.52,A -85,B 0,C 180,E1 -11757.875,E2 -11757.875} C_VEL
LIN {X 0,Y 390.091,Z 350.538,A -85,B 0,C 180,E1 -11760.086,E2 -11760.086} C_VEL
LIN {X 0,Y 390.88,Z 353.776,A -85,B 0,C 180,E1 -11760.956,E2 -11760.956} C_VEL
LIN {X 0,Y 393.498,Z 365.541,A -85,B 0,C 180,E1 -11763.765,E2 -11763.765} C_VEL
LIN {X 0,Y 394.708,Z 372.174,A -85,B 0,C 180,E1 -11765.242,E2 -11765.242} C_VEL
LIN {X 0,Y 396.03,Z 378.122,A -85,B 0,C 180,E1 -11765.487,E2 -11765.487} C_VEL
LIN {X 0,Y 400.903,Z 403.089,A -85,B 0,C 180,E1 -11766.284,E2 -11766.284} C_VEL
LIN {X 0,Y 399.034,Z 509.303,A -85,B 0,C 180,E1 -11768.224,E2 -11768.224} C_VEL
LIN {X 0,Y 398.364,Z 523.236,A -85,B 0,C 180,E1 -11768.661,E2 -11768.661} C_VEL
LIN {X 0,Y 397.58,Z 536.856,A -85,B 0,C 180,E1 -11769.295,E2 -11769.295} C_VEL
LIN {X 0,Y 396.729,Z 548.781,A -85,B 0,C 180,E1 -11770.028,E2 -11770.028} C_VEL
LIN {X 0,Y 395.659,Z 560.708,A -85,B 0,C 180,E1 -11770.949,E2 -11770.949} C_VEL
LIN {X 0,Y 394.447,Z 572.688,A -85,B 0,C 180,E1 -11772.099,E2 -11772.099} C_VEL
LIN {X 0,Y 393.743,Z 578.997,A -85,B 0,C 180,E1 -11772.81,E2 -11772.81} C_VEL
LIN {X 0,Y 392.66,Z 583.548,A -85,B 0,C 180,E1 -11773.347,E2 -11773.347} C_VEL
LIN {X 0,Y 389.03,Z 590.641,A -85,B 0,C 180,E1 -11774.213,E2 -11774.213} C_VEL
LIN {X 0,Y 385.412,Z 597.305,A -85,B 0,C 180,E1 -11775.159,E2 -11775.159} C_VEL
LIN {X 0,Y 384.36,Z 601.086,A -85,B 0,C 180,E1 -11775.812,E2 -11775.812} C_VEL
LIN {X 0,Y 383.5,Z 609.591,A -85,B 0,C 180,E1 -11777.564,E2 -11777.564} C_VEL
LIN {X 0,Y 382.709,Z 616.883,A -85,B 0,C 180,E1 -11779.417,E2 -11779.417} C_VEL
LIN {X 0,Y 382.078,Z 623.434,A -85,B 0,C 180,E1 -11781.537,E2 -11781.537} C_VEL
LIN {X 0,Y 381.766,Z 628.342,A -85,B 0,C 180,E1 -11783.657,E2 -11783.657} C_VEL
LIN {X 0,Y 381.627,Z 631.762,A -85,B 0,C 180,E1 -11785.774,E2 -11785.774} C_VEL
LIN {X 0,Y 381.516,Z 633.798,A -85,B 0,C 180,E1 -11787.887,E2 -11787.887} C_VEL
LIN {X 0,Y 381.54,Z 634.498,A -85,B 0,C 180,E1 -11789.999,E2 -11789.999} C_VEL
LIN {X 0,Y 381.515,Z 633.871,A -85,B 0,C 180,E1 -11792.11,E2 -11792.11} C_VEL
LIN {X 0,Y 381.624,Z 631.905,A -85,B 0,C 180,E1 -11794.223,E2 -11794.223} C_VEL
LIN {X 0,Y 381.766,Z 628.548,A -85,B 0,C 180,E1 -11796.34,E2 -11796.34} C_VEL
LIN {X 0,Y 382.072,Z 623.703,A -85,B 0,C 180,E1 -11798.461,E2 -11798.461} C_VEL
LIN {X 0,Y 382.509,Z 619.033,A -85,B 0,C 180,E1 -11800.051,E2 -11800.051} C_VEL
LIN {X 0,Y 383.206,Z 612.246,A -85,B 0,C 180,E1 -11801.906,E2 -11801.906} C_VEL
LIN {X 0,Y 383.975,Z 605.161,A -85,B 0,C 180,E1 -11803.494,E2 -11803.494} C_VEL
LIN {X 0,Y 384.948,Z 596.635,A -85,B 0,C 180,E1 -11805.078,E2 -11805.078} C_VEL
LIN {X 0,Y 386.112,Z 586.303,A -85,B 0,C 180,E1 -11806.658,E2 -11806.658} C_VEL
LIN {X 0,Y 387.452,Z 574.746,A -85,B 0,C 180,E1 -11808.096,E2 -11808.096} C_VEL
LIN {X 0,Y 388.663,Z 563.209,A -85,B 0,C 180,E1 -11809.268,E2 -11809.268} C_VEL
LIN {X 0,Y 389.96,Z 549.796,A -85,B 0,C 180,E1 -11810.355,E2 -11810.355} C_VEL
LIN {X 0,Y 390.978,Z 536.279,A -85,B 0,C 180,E1 -11811.206,E2 -11811.206} C_VEL
LIN {X 0,Y 391.862,Z 522.441,A -85,B 0,C 180,E1 -11811.847,E2 -11811.847} C_VEL
LIN {X 0,Y 392.546,Z 507.872,A -85,B 0,C 180,E1 -11812.291,E2 -11812.291} C_VEL
LIN {X 0,Y 394.449,Z 404.089,A -85,B 0,C 180,E1 -11814.21,E2 -11814.21} C_VEL
LIN {X 0,Y 390.399,Z 383.291,A -85,B 0,C 180,E1 -11814.89,E2 -11814.89} C_VEL
LIN {X 0,Y 388.122,Z 373.78,A -85,B 0,C 180,E1 -11815.237,E2 -11815.237} C_VEL
LIN {X 0,Y 387.546,Z 371.874,A -85,B 0,C 180,E1 -11815.394,E2 -11815.394} C_VEL
LIN {X 0,Y 384.985,Z 359.479,A -85,B 0,C 180,E1 -11818.334,E2 -11818.334} C_VEL
LIN {X 0,Y 383.045,Z 351.7,A -85,B 0,C 180,E1 -11820.306,E2 -11820.306} C_VEL
LIN {X 0,Y 383.005,Z 351.385,A -85,B 0,C 180,E1 -11820.611,E2 -11820.611} C_VEL
LIN {X 0,Y 383.012,Z 351.395,A -85,B 0,C 180,E1 -11823.398,E2 -11823.398} C_VEL
LIN {X 0,Y 383.029,Z 351.388,A -85,B 0,C 180,E1 -11826.164,E2 -11826.164} C_VEL
LIN {X 0,Y 383.016,Z 351.385,A -85,B 0,C 180,E1 -11829.955,E2 -11829.955} C_VEL
LIN {X 0,Y 383.06,Z 351.393,A -85,B 0,C 180,E1 -11832.787,E2 -11832.787} C_VEL
LIN {X 0,Y 383.066,Z 351.372,A -85,B 0,C 180,E1 -11835.799,E2 -11835.799} C_VEL
LIN {X 0,Y 383.037,Z 351.396,A -85,B 0,C 180,E1 -11838.785,E2 -11838.785} C_VEL
LIN {X 0,Y 382.996,Z 351.37,A -85,B 0,C 180,E1 -11842.094,E2 -11842.094} C_VEL
LIN {X 0,Y 383.01,Z 351.397,A -85,B 0,C 180,E1 -11845.331,E2 -11845.331} C_VEL
LIN {X 0,Y 382.977,Z 351.382,A -85,B 0,C 180,E1 -11849.081,E2 -11849.081} C_VEL
LIN {X 0,Y 383.047,Z 351.372,A -85,B 0,C 180,E1 -11852.697,E2 -11852.697} C_VEL
LIN {X 0,Y 383.024,Z 351.397,A -85,B 0,C 180,E1 -11856.192,E2 -11856.192} C_VEL
LIN {X 0,Y 383.045,Z 351.388,A -85,B 0,C 180,E1 -11859.598,E2 -11859.598} C_VEL
LIN {X 0,Y 383.094,Z 351.388,A -85,B 0,C 180,E1 -11862.931,E2 -11862.931} C_VEL
LIN {X 0,Y 383.115,Z 351.381,A -85,B 0,C 180,E1 -11866.463,E2 -11866.463} C_VEL
LIN {X 0,Y 383.131,Z 351.373,A -85,B 0,C 180,E1 -11869.43,E2 -11869.43} C_VEL
LIN {X 0,Y 383.263,Z 351.363,A -85,B 0,C 180,E1 -11872.625,E2 -11872.625} C_VEL
LIN {X 0,Y 383.192,Z 351.377,A -85,B 0,C 180,E1 -11874.738,E2 -11874.738} C_VEL
LIN {X 0,Y 383.378,Z 351.347,A -85,B 0,C 180,E1 -11877.899,E2 -11877.899} C_VEL
LIN {X 0,Y 383.513,Z 351.336,A -85,B 0,C 180,E1 -11880,E2 -11880} C_VEL
LIN {X 0,Y 383.244,Z 351.357,A -85,B 0,C 180,E1 -11883.154,E2 -11883.154} C_VEL
LIN {X 0,Y 383.278,Z 351.364,A -85,B 0,C 180,E1 -11886.316,E2 -11886.316} C_VEL
LIN {X 0,Y 383.25,Z 351.363,A -85,B 0,C 180,E1 -11888.436,E2 -11888.436} C_VEL
LIN {X 0,Y 383.098,Z 351.384,A -85,B 0,C 180,E1 -11891.642,E2 -11891.642} C_VEL
LIN {X 0,Y 383.101,Z 351.375,A -85,B 0,C 180,E1 -11894.882,E2 -11894.882} C_VEL
LIN {X 0,Y 383.078,Z 351.388,A -85,B 0,C 180,E1 -11898.173,E2 -11898.173} C_VEL
LIN {X 0,Y 382.986,Z 351.39,A -85,B 0,C 180,E1 -11901.531,E2 -11901.531} C_VEL
LIN {X 0,Y 383.043,Z 351.392,A -85,B 0,C 180,E1 -11904.961,E2 -11904.961} C_VEL
LIN {X 0,Y 383.007,Z 351.359,A -85,B 0,C 180,E1 -11908.495,E2 -11908.495} C_VEL
LIN {X 0,Y 382.999,Z 351.393,A -85,B 0,C 180,E1 -11912.151,E2 -11912.151} C_VEL
LIN {X 0,Y 383.009,Z 351.397,A -85,B 0,C 180,E1 -11914.669,E2 -11914.669} C_VEL
LIN {X 0,Y 382.995,Z 351.37,A -85,B 0,C 180,E1 -11917.906,E2 -11917.906} C_VEL
LIN {X 0,Y 383.039,Z 351.395,A -85,B 0,C 180,E1 -11921.34,E2 -11921.34} C_VEL
LIN {X 0,Y 383.063,Z 351.372,A -85,B 0,C 180,E1 -11924.316,E2 -11924.316} C_VEL
LIN {X 0,Y 383.068,Z 351.392,A -85,B 0,C 180,E1 -11927.25,E2 -11927.25} C_VEL
LIN {X 0,Y 383.016,Z 351.386,A -85,B 0,C 180,E1 -11930.413,E2 -11930.413} C_VEL
LIN {X 0,Y 383.021,Z 351.389,A -85,B 0,C 180,E1 -11934.046,E2 -11934.046} C_VEL
LIN {X 0,Y 383.033,Z 351.392,A -85,B 0,C 180,E1 -11937.854,E2 -11937.854} C_VEL
LIN {X 0,Y 383.044,Z 351.572,A -85,B 0,C 180,E1 -11939.694,E2 -11939.694} C_VEL
LIN {X 0,Y 385.53,Z 361.895,A -85,B 0,C 180,E1 -11942.301,E2 -11942.301} C_VEL
LIN {X 0,Y 387.611,Z 372.149,A -85,B 0,C 180,E1 -11944.699,E2 -11944.699} C_VEL
LIN {X 0,Y 389.014,Z 376.586,A -85,B 0,C 180,E1 -11944.927,E2 -11944.927} C_VEL
LIN {X 0,Y 394.286,Z 402.808,A -85,B 0,C 180,E1 -11945.799,E2 -11945.799} C_VEL
LIN {X 0,Y 394.123,Z 424.18,A -85,B 0,C 180,E1 -11946.206,E2 -11946.206} C_VEL
LIN {X 0,Y 392.448,Z 510.105,A -85,B 0,C 180,E1 -11947.807,E2 -11947.807} C_VEL
LIN {X 0,Y 391.742,Z 524.517,A -85,B 0,C 180,E1 -11948.285,E2 -11948.285} C_VEL
LIN {X 0,Y 390.893,Z 537.802,A -85,B 0,C 180,E1 -11948.927,E2 -11948.927} C_VEL
LIN {X 0,Y 389.822,Z 551.629,A -85,B 0,C 180,E1 -11949.825,E2 -11949.825} C_VEL
LIN {X 0,Y 388.647,Z 564.167,A -85,B 0,C 180,E1 -11950.869,E2 -11950.869} C_VEL
LIN {X 0,Y 387.229,Z 576.703,A -85,B 0,C 180,E1 -11952.167,E2 -11952.167} C_VEL
LIN {X 0,Y 385.938,Z 587.871,A -85,B 0,C 180,E1 -11953.607,E2 -11953.607} C_VEL
LIN {X 0,Y 384.707,Z 597.885,A -85,B 0,C 180,E1 -11955.183,E2 -11955.183} C_VEL
LIN {X 0,Y 383.931,Z 606.201,A -85,B 0,C 180,E1 -11956.774,E2 -11956.774} C_VEL
LIN {X 0,Y 382.951,Z 614.148,A -85,B 0,C 180,E1 -11958.623,E2 -11958.623} C_VEL
LIN {X 0,Y 382.349,Z 620.543,A -85,B 0,C 180,E1 -11960.479,E2 -11960.479} C_VEL
LIN {X 0,Y 381.859,Z 626.214,A -85,B 0,C 180,E1 -11962.599,E2 -11962.599} C_VEL
LIN {X 0,Y 381.802,Z 628.58,A -85,B 0,C 180,E1 -11963.721,E2 -11963.721} C_VEL
LIN {X 0,Y 381.626,Z 631.843,A -85,B 0,C 180,E1 -11965.777,E2 -11965.777} C_VEL
LIN {X 0,Y 381.514,Z 633.841,A -85,B 0,C 180,E1 -11967.89,E2 -11967.89} C_VEL
LIN {X 0,Y 381.539,Z 634.5,A -85,B 0,C 180,E1 -11970.001,E2 -11970.001} C_VEL
LIN {X 0,Y 381.515,Z 633.831,A -85,B 0,C 180,E1 -11972.113,E2 -11972.113} C_VEL
LIN {X 0,Y 381.625,Z 631.824,A -85,B 0,C 180,E1 -11974.226,E2 -11974.226} C_VEL
LIN {X 0,Y 381.765,Z 628.432,A -85,B 0,C 180,E1 -11976.343,E2 -11976.343} C_VEL
LIN {X 0,Y 382.073,Z 623.554,A -85,B 0,C 180,E1 -11978.463,E2 -11978.463} C_VEL
LIN {X 0,Y 382.516,Z 618.844,A -85,B 0,C 180,E1 -11980.053,E2 -11980.053} C_VEL
LIN {X 0,Y 383.224,Z 612.01,A -85,B 0,C 180,E1 -11981.908,E2 -11981.908} C_VEL
LIN {X 0,Y 384.023,Z 604.88,A -85,B 0,C 180,E1 -11983.495,E2 -11983.495} C_VEL
LIN {X 0,Y 384.906,Z 596.297,A -85,B 0,C 180,E1 -11985.083,E2 -11985.083} C_VEL
LIN {X 0,Y 386.153,Z 585.892,A -85,B 0,C 180,E1 -11986.659,E2 -11986.659} C_VEL
LIN {X 0,Y 387.339,Z 575.426,A -85,B 0,C 180,E1 -11987.967,E2 -11987.967} C_VEL
LIN {X 0,Y 388.622,Z 564.032,A -85,B 0,C 180,E1 -11989.135,E2 -11989.135} C_VEL
LIN {X 0,Y 389.807,Z 550.993,A -85,B 0,C 180,E1 -11990.215,E2 -11990.215} C_VEL
LIN {X 0,Y 390.875,Z 537.601,A -85,B 0,C 180,E1 -11991.077,E2 -11991.077} C_VEL
LIN {X 0,Y 391.735,Z 524.239,A -85,B 0,C 180,E1 -11991.718,E2 -11991.718} C_VEL
LIN {X 0,Y 392.387,Z 510.814,A -85,B 0,C 180,E1 -11992.165,E2 -11992.165} C_VEL
LIN {X 0,Y 393.093,Z 480.816,A -85,B 0,C 180,E1 -11992.746,E2 -11992.746} C_VEL
LIN {X 0,Y 394.335,Z 403.281,A -85,B 0,C 180,E1 -11994.178,E2 -11994.178} C_VEL
LIN {X 0,Y 389.346,Z 378.133,A -85,B 0,C 180,E1 -11995.021,E2 -11995.021} C_VEL
LIN {X 0,Y 389.291,Z 376.02,A -85,B 0,C 180,E1 -11995.203,E2 -11995.203} C_VEL
LIN {X 0,Y 386.559,Z 366.798,A -85,B 0,C 180,E1 -11996.549,E2 -11996.549} C_VEL
LIN {X 0,Y 383.963,Z 355.154,A -85,B 0,C 180,E1 -11999.347,E2 -11999.347} C_VEL
LIN {X 0,Y 383.027,Z 351.532,A -85,B 0,C 180,E1 -12000.308,E2 -12000.308} C_VEL
LIN {X 0,Y 383.016,Z 351.4,A -85,B 0,C 180,E1 -12003.401,E2 -12003.401} C_VEL
LIN {X 0,Y 383.038,Z 351.396,A -85,B 0,C 180,E1 -12006.166,E2 -12006.166} C_VEL
LIN {X 0,Y 383.013,Z 351.4,A -85,B 0,C 180,E1 -12009.959,E2 -12009.959} C_VEL
LIN {X 0,Y 383.01,Z 351.398,A -85,B 0,C 180,E1 -12012.779,E2 -12012.779} C_VEL
LIN {X 0,Y 383.002,Z 351.403,A -85,B 0,C 180,E1 -12015.79,E2 -12015.79} C_VEL
LIN {X 0,Y 382.993,Z 351.405,A -85,B 0,C 180,E1 -12018.796,E2 -12018.796} C_VEL
LIN {X 0,Y 383.004,Z 351.402,A -85,B 0,C 180,E1 -12022.097,E2 -12022.097} C_VEL
LIN {X 0,Y 383.06,Z 351.64,A -85,B 0,C 180,E1 -12023.713,E2 -12023.713} C_VEL
LIN {X 0,Y 385.831,Z 358.654,A -85,B 0,C 180,E1 -12025.819,E2 -12025.819} C_VEL
LIN {X 0,Y 388.398,Z 366.036,A -85,B 0,C 180,E1 -12027.738,E2 -12027.738} C_VEL
LIN {X 0,Y 390.848,Z 374.743,A -85,B 0,C 180,E1 -12029.77,E2 -12029.77} C_VEL
LIN {X 0,Y 392.295,Z 382.436,A -85,B 0,C 180,E1 -12031.385,E2 -12031.385} C_VEL
LIN {X 0,Y 390.845,Z 399.301,A -85,B 0,C 180,E1 -12034.219,E2 -12034.219} C_VEL
LIN {X 0,Y 389.102,Z 420.443,A -85,B 0,C 180,E1 -12037.664,E2 -12037.664} C_VEL
LIN {X 0,Y 392.078,Z 435.409,A -85,B 0,C 180,E1 -12038.451,E2 -12038.451} C_VEL
LIN {X 0,Y 393.462,Z 446.828,A -85,B 0,C 180,E1 -12038.938,E2 -12038.938} C_VEL
LIN {X 0,Y 390.708,Z 514.122,A -85,B 0,C 180,E1 -12040.733,E2 -12040.733} C_VEL
LIN {X 0,Y 389.941,Z 534.578,A -85,B 0,C 180,E1 -12041.308,E2 -12041.308} C_VEL
LIN {X 0,Y 389.168,Z 547.121,A -85,B 0,C 180,E1 -12041.849,E2 -12041.849} C_VEL
LIN {X 0,Y 388.213,Z 560.09,A -85,B 0,C 180,E1 -12042.62,E2 -12042.62} C_VEL
LIN {X 0,Y 387.128,Z 573.182,A -85,B 0,C 180,E1 -12043.657,E2 -12043.657} C_VEL
LIN {X 0,Y 386.034,Z 584.315,A -85,B 0,C 180,E1 -12044.778,E2 -12044.778} C_VEL
LIN {X 0,Y 385.064,Z 594.157,A -85,B 0,C 180,E1 -12046.005,E2 -12046.005} C_VEL
LIN {X 0,Y 384.157,Z 602.843,A -85,B 0,C 180,E1 -12047.318,E2 -12047.318} C_VEL
LIN {X 0,Y 383.372,Z 611.297,A -85,B 0,C 180,E1 -12048.902,E2 -12048.902} C_VEL
LIN {X 0,Y 382.719,Z 618.118,A -85,B 0,C 180,E1 -12050.487,E2 -12050.487} C_VEL
LIN {X 0,Y 382.183,Z 623.562,A -85,B 0,C 180,E1 -12052.073,E2 -12052.073} C_VEL
LIN {X 0,Y 381.872,Z 627.773,A -85,B 0,C 180,E1 -12053.66,E2 -12053.66} C_VEL
LIN {X 0,Y 381.799,Z 629.952,A -85,B 0,C 180,E1 -12054.719,E2 -12054.719} C_VEL
LIN {X 0,Y 381.658,Z 631.662,A -85,B 0,C 180,E1 -12055.776,E2 -12055.776} C_VEL
LIN {X 0,Y 381.54,Z 632.95,A -85,B 0,C 180,E1 -12056.832,E2 -12056.832} C_VEL
LIN {X 0,Y 381.537,Z 633.772,A -85,B 0,C 180,E1 -12057.889,E2 -12057.889} C_VEL
LIN {X 0,Y 381.557,Z 634.151,A -85,B 0,C 180,E1 -12058.945,E2 -12058.945} C_VEL
LIN {X 0,Y 381.543,Z 634.115,A -85,B 0,C 180,E1 -12060,E2 -12060} C_VEL
LIN {X 0,Y 381.556,Z 633.634,A -85,B 0,C 180,E1 -12061.055,E2 -12061.055} C_VEL
LIN {X 0,Y 381.52,Z 632.686,A -85,B 0,C 180,E1 -12062.111,E2 -12062.111} C_VEL
LIN {X 0,Y 381.528,Z 631.318,A -85,B 0,C 180,E1 -12063.168,E2 -12063.168} C_VEL
LIN {X 0,Y 381.682,Z 628.388,A -85,B 0,C 180,E1 -12064.753,E2 -12064.753} C_VEL
LIN {X 0,Y 381.771,Z 624.344,A -85,B 0,C 180,E1 -12066.342,E2 -12066.342} C_VEL
LIN {X 0,Y 382.062,Z 618.029,A -85,B 0,C 180,E1 -12068.196,E2 -12068.196} C_VEL
LIN {X 0,Y 382.421,Z 611.101,A -85,B 0,C 180,E1 -12069.788,E2 -12069.788} C_VEL
LIN {X 0,Y 382.846,Z 604.01,A -85,B 0,C 180,E1 -12071.113,E2 -12071.113} C_VEL
LIN {X 0,Y 383.465,Z 595.434,A -85,B 0,C 180,E1 -12072.436,E2 -12072.436} C_VEL
LIN {X 0,Y 384.182,Z 584.908,A -85,B 0,C 180,E1 -12073.758,E2 -12073.758} C_VEL
LIN {X 0,Y 384.77,Z 574.557,A -85,B 0,C 180,E1 -12074.816,E2 -12074.816} C_VEL
LIN {X 0,Y 385.42,Z 563.228,A -85,B 0,C 180,E1 -12075.738,E2 -12075.738} C_VEL
LIN {X 0,Y 386.125,Z 549.587,A -85,B 0,C 180,E1 -12076.591,E2 -12076.591} C_VEL
LIN {X 0,Y 386.716,Z 536.239,A -85,B 0,C 180,E1 -12077.177,E2 -12077.177} C_VEL
LIN {X 0,Y 387.04,Z 522.398,A -85,B 0,C 180,E1 -12077.571,E2 -12077.571} C_VEL
LIN {X 0,Y 388.689,Z 444.643,A -85,B 0,C 180,E1 -12079.384,E2 -12079.384} C_VEL
LIN {X 0,Y 385.629,Z 420.6,A -85,B 0,C 180,E1 -12080.116,E2 -12080.116} C_VEL
LIN {X 0,Y 386.848,Z 398.954,A -85,B 0,C 180,E1 -12083.558,E2 -12083.558} C_VEL
LIN {X 0,Y 388.189,Z 376.858,A -85,B 0,C 180,E1 -12087.108,E2 -12087.108} C_VEL
LIN {X 0,Y 387.744,Z 372.189,A -85,B 0,C 180,E1 -12087.902,E2 -12087.902} C_VEL
LIN {X 0,Y 383.572,Z 353.96,A -85,B 0,C 180,E1 -12091.172,E2 -12091.172} C_VEL
LIN {X 0,Y 383.03,Z 351.498,A -85,B 0,C 180,E1 -12091.684,E2 -12091.684} C_VEL
LIN {X 0,Y 383.024,Z 351.402,A -85,B 0,C 180,E1 -12094.668,E2 -12094.668} C_VEL
LIN {X 0,Y 383.004,Z 351.402,A -85,B 0,C 180,E1 -12097.903,E2 -12097.903} C_VEL
LIN {X 0,Y 382.989,Z 351.401,A -85,B 0,C 180,E1 -12101.347,E2 -12101.347} C_VEL
LIN {X 0,Y 383.001,Z 351.38,A -85,B 0,C 180,E1 -12104.303,E2 -12104.303} C_VEL
LIN {X 0,Y 383.016,Z 351.399,A -85,B 0,C 180,E1 -12107.24,E2 -12107.24} C_VEL
LIN {X 0,Y 383.021,Z 351.385,A -85,B 0,C 180,E1 -12110.413,E2 -12110.413} C_VEL
LIN {X 0,Y 383.032,Z 351.388,A -85,B 0,C 180,E1 -12114.044,E2 -12114.044} C_VEL
LIN {X 0,Y 382.992,Z 351.395,A -85,B 0,C 180,E1 -12117.577,E2 -12117.577} C_VEL
LIN {X 0,Y 383.045,Z 351.576,A -85,B 0,C 180,E1 -12119.762,E2 -12119.762} C_VEL
LIN {X 0,Y 385.44,Z 361.622,A -85,B 0,C 180,E1 -12122.291,E2 -12122.291} C_VEL
LIN {X 0,Y 387.594,Z 372.114,A -85,B 0,C 180,E1 -12124.747,E2 -12124.747} C_VEL
LIN {X 0,Y 388.975,Z 376.526,A -85,B 0,C 180,E1 -12124.98,E2 -12124.98} C_VEL
LIN {X 0,Y 394.366,Z 403.272,A -85,B 0,C 180,E1 -12125.869,E2 -12125.869} C_VEL
LIN {X 0,Y 392.469,Z 509.32,A -85,B 0,C 180,E1 -12127.84,E2 -12127.84} C_VEL
LIN {X 0,Y 391.759,Z 523.247,A -85,B 0,C 180,E1 -12128.283,E2 -12128.283} C_VEL
LIN {X 0,Y 390.947,Z 536.864,A -85,B 0,C 180,E1 -12128.927,E2 -12128.927} C_VEL
LIN {X 0,Y 389.987,Z 549.503,A -85,B 0,C 180,E1 -12129.723,E2 -12129.723} C_VEL
LIN {X 0,Y 388.798,Z 562.139,A -85,B 0,C 180,E1 -12130.737,E2 -12130.737} C_VEL
LIN {X 0,Y 387.518,Z 573.866,A -85,B 0,C 180,E1 -12131.905,E2 -12131.905} C_VEL
LIN {X 0,Y 386.22,Z 585.57,A -85,B 0,C 180,E1 -12133.344,E2 -12133.344} C_VEL
LIN {X 0,Y 384.96,Z 596.027,A -85,B 0,C 180,E1 -12134.92,E2 -12134.92} C_VEL
LIN {X 0,Y 384.36,Z 601.086,A -85,B 0,C 180,E1 -12135.812,E2 -12135.812} C_VEL
LIN {X 0,Y 383.35,Z 604.713,A -85,B 0,C 180,E1 -12136.493,E2 -12136.493} C_VEL
LIN {X 0,Y 379.901,Z 610.284,A -85,B 0,C 180,E1 -12137.613,E2 -12137.613} C_VEL
LIN {X 0,Y 376.49,Z 615.349,A -85,B 0,C 180,E1 -12138.803,E2 -12138.803} C_VEL
LIN {X 0,Y 375.555,Z 618.115,A -85,B 0,C 180,E1 -12139.584,E2 -12139.584} C_VEL
LIN {X 0,Y 375.024,Z 623.435,A -85,B 0,C 180,E1 -12141.376,E2 -12141.376} C_VEL
LIN {X 0,Y 374.679,Z 628.343,A -85,B 0,C 180,E1 -12143.537,E2 -12143.537} C_VEL
LIN {X 0,Y 374.556,Z 631.763,A -85,B 0,C 180,E1 -12145.694,E2 -12145.694} C_VEL
LIN {X 0,Y 374.416,Z 633.798,A -85,B 0,C 180,E1 -12147.847,E2 -12147.847} C_VEL
LIN {X 0,Y 374.441,Z 634.498,A -85,B 0,C 180,E1 -12149.999,E2 -12149.999} C_VEL
LIN {X 0,Y 374.415,Z 633.871,A -85,B 0,C 180,E1 -12152.15,E2 -12152.15} C_VEL
LIN {X 0,Y 374.552,Z 631.904,A -85,B 0,C 180,E1 -12154.303,E2 -12154.303} C_VEL
LIN {X 0,Y 374.681,Z 628.547,A -85,B 0,C 180,E1 -12156.461,E2 -12156.461} C_VEL
LIN {X 0,Y 375.017,Z 623.701,A -85,B 0,C 180,E1 -12158.621,E2 -12158.621} C_VEL
LIN {X 0,Y 375.471,Z 619.032,A -85,B 0,C 180,E1 -12160.241,E2 -12160.241} C_VEL
LIN {X 0,Y 376.246,Z 612.244,A -85,B 0,C 180,E1 -12162.129,E2 -12162.129} C_VEL
LIN {X 0,Y 377.012,Z 605.159,A -85,B 0,C 180,E1 -12163.748,E2 -12163.748} C_VEL
LIN {X 0,Y 378.054,Z 596.632,A -85,B 0,C 180,E1 -12165.36,E2 -12165.36} C_VEL
LIN {X 0,Y 379.275,Z 586.299,A -85,B 0,C 180,E1 -12166.967,E2 -12166.967} C_VEL
LIN {X 0,Y 380.685,Z 574.742,A -85,B 0,C 180,E1 -12168.429,E2 -12168.429} C_VEL
LIN {X 0,Y 381.966,Z 563.204,A -85,B 0,C 180,E1 -12169.619,E2 -12169.619} C_VEL
LIN {X 0,Y 383.3,Z 549.842,A -85,B 0,C 180,E1 -12170.721,E2 -12170.721} C_VEL
LIN {X 0,Y 384.378,Z 536.271,A -85,B 0,C 180,E1 -12171.589,E2 -12171.589} C_VEL
LIN {X 0,Y 385.267,Z 522.43,A -85,B 0,C 180,E1 -12172.24,E2 -12172.24} C_VEL
LIN {X 0,Y 385.991,Z 507.85,A -85,B 0,C 180,E1 -12172.69,E2 -12172.69} C_VEL
LIN {X 0,Y 387.937,Z 404.463,A -85,B 0,C 180,E1 -12174.636,E2 -12174.636} C_VEL
LIN {X 0,Y 382.621,Z 378.259,A -85,B 0,C 180,E1 -12175.533,E2 -12175.533} C_VEL
LIN {X 0,Y 380.434,Z 372.189,A -85,B 0,C 180,E1 -12175.855,E2 -12175.855} C_VEL
LIN {X 0,Y 378.035,Z 360.784,A -85,B 0,C 180,E1 -12178.6,E2 -12178.6} C_VEL
LIN {X 0,Y 375.975,Z 352.343,A -85,B 0,C 180,E1 -12180.835,E2 -12180.835} C_VEL
LIN {X 0,Y 375.976,Z 352.276,A -85,B 0,C 180,E1 -12184.666,E2 -12184.666} C_VEL
LIN {X 0,Y 375.973,Z 352.276,A -85,B 0,C 180,E1 -12188.27,E2 -12188.27} C_VEL
LIN {X 0,Y 375.984,Z 352.272,A -85,B 0,C 180,E1 -12191.609,E2 -12191.609} C_VEL
LIN {X 0,Y 376.01,Z 352.248,A -85,B 0,C 180,E1 -12195.253,E2 -12195.253} C_VEL
LIN {X 0,Y 375.993,Z 352.274,A -85,B 0,C 180,E1 -12199.14,E2 -12199.14} C_VEL
LIN {X 0,Y 375.96,Z 352.246,A -85,B 0,C 180,E1 -12201.911,E2 -12201.911} C_VEL
LIN {X 0,Y 375.971,Z 352.274,A -85,B 0,C 180,E1 -12205.331,E2 -12205.331} C_VEL
LIN {X 0,Y 375.951,Z 352.268,A -85,B 0,C 180,E1 -12208.437,E2 -12208.437} C_VEL
LIN {X 0,Y 375.993,Z 352.239,A -85,B 0,C 180,E1 -12212.141,E2 -12212.141} C_VEL
LIN {X 0,Y 375.997,Z 352.268,A -85,B 0,C 180,E1 -12214.538,E2 -12214.538} C_VEL
LIN {X 0,Y 375.954,Z 352.268,A -85,B 0,C 180,E1 -12218.045,E2 -12218.045} C_VEL
LIN {X 0,Y 376.014,Z 352.273,A -85,B 0,C 180,E1 -12221.473,E2 -12221.473} C_VEL
LIN {X 0,Y 376.049,Z 352.251,A -85,B 0,C 180,E1 -12224.832,E2 -12224.832} C_VEL
LIN {X 0,Y 376.049,Z 352.262,A -85,B 0,C 180,E1 -12228.136,E2 -12228.136} C_VEL
LIN {X 0,Y 376.247,Z 352.236,A -85,B 0,C 180,E1 -12231.877,E2 -12231.877} C_VEL
LIN {X 0,Y 376.164,Z 352.251,A -85,B 0,C 180,E1 -12234.64,E2 -12234.64} C_VEL
LIN {X 0,Y 376.344,Z 352.223,A -85,B 0,C 180,E1 -12237.859,E2 -12237.859} C_VEL
LIN {X 0,Y 376.482,Z 352.212,A -85,B 0,C 180,E1 -12240,E2 -12240} C_VEL
LIN {X 0,Y 376.182,Z 352.236,A -85,B 0,C 180,E1 -12243.213,E2 -12243.213} C_VEL
LIN {X 0,Y 376.237,Z 352.242,A -85,B 0,C 180,E1 -12246.435,E2 -12246.435} C_VEL
LIN {X 0,Y 376.195,Z 352.238,A -85,B 0,C 180,E1 -12248.595,E2 -12248.595} C_VEL
LIN {X 0,Y 376.049,Z 352.261,A -85,B 0,C 180,E1 -12251.863,E2 -12251.863} C_VEL
LIN {X 0,Y 376.049,Z 352.25,A -85,B 0,C 180,E1 -12255.168,E2 -12255.168} C_VEL
LIN {X 0,Y 376.014,Z 352.271,A -85,B 0,C 180,E1 -12258.526,E2 -12258.526} C_VEL
LIN {X 0,Y 375.955,Z 352.267,A -85,B 0,C 180,E1 -12261.955,E2 -12261.955} C_VEL
LIN {X 0,Y 375.997,Z 352.267,A -85,B 0,C 180,E1 -12265.462,E2 -12265.462} C_VEL
LIN {X 0,Y 375.973,Z 352.233,A -85,B 0,C 180,E1 -12268.534,E2 -12268.534} C_VEL
LIN {X 0,Y 375.948,Z 352.268,A -85,B 0,C 180,E1 -12271.563,E2 -12271.563} C_VEL
LIN {X 0,Y 375.949,Z 352.273,A -85,B 0,C 180,E1 -12275.416,E2 -12275.416} C_VEL
LIN {X 0,Y 375.969,Z 352.245,A -85,B 0,C 180,E1 -12278.272,E2 -12278.272} C_VEL
LIN {X 0,Y 375.982,Z 352.276,A -85,B 0,C 180,E1 -12281.611,E2 -12281.611} C_VEL
LIN {X 0,Y 376.009,Z 352.25,A -85,B 0,C 180,E1 -12285.256,E2 -12285.256} C_VEL
LIN {X 0,Y 375.983,Z 352.273,A -85,B 0,C 180,E1 -12288.391,E2 -12288.391} C_VEL
LIN {X 0,Y 375.962,Z 352.278,A -85,B 0,C 180,E1 -12291.913,E2 -12291.913} C_VEL
LIN {X 0,Y 375.975,Z 352.276,A -85,B 0,C 180,E1 -12295.334,E2 -12295.334} C_VEL
LIN {X 0,Y 375.967,Z 352.33,A -85,B 0,C 180,E1 -12299.199,E2 -12299.199} C_VEL
LIN {X 0,Y 377.637,Z 359.048,A -85,B 0,C 180,E1 -12301.009,E2 -12301.009} C_VEL
LIN {X 0,Y 379.967,Z 369.741,A -85,B 0,C 180,E1 -12303.648,E2 -12303.648} C_VEL
LIN {X 0,Y 380.518,Z 372.353,A -85,B 0,C 180,E1 -12304.212,E2 -12304.212} C_VEL
LIN {X 0,Y 382.857,Z 379.055,A -85,B 0,C 180,E1 -12304.545,E2 -12304.545} C_VEL
LIN {X 0,Y 387.851,Z 403.86,A -85,B 0,C 180,E1 -12305.392,E2 -12305.392} C_VEL
LIN {X 0,Y 386.582,Z 479.734,A -85,B 0,C 180,E1 -12306.816,E2 -12306.816} C_VEL
LIN {X 0,Y 385.902,Z 510.118,A -85,B 0,C 180,E1 -12307.41,E2 -12307.41} C_VEL
LIN {X 0,Y 385.149,Z 524.525,A -85,B 0,C 180,E1 -12307.894,E2 -12307.894} C_VEL
LIN {X 0,Y 384.27,Z 537.808,A -85,B 0,C 180,E1 -12308.546,E2 -12308.546} C_VEL
LIN {X 0,Y 383.165,Z 551.442,A -85,B 0,C 180,E1 -12309.443,E2 -12309.443} C_VEL
LIN {X 0,Y 381.918,Z 564.171,A -85,B 0,C 180,E1 -12310.518,E2 -12310.518} C_VEL
LIN {X 0,Y 380.432,Z 576.706,A -85,B 0,C 180,E1 -12311.837,E2 -12311.837} C_VEL
LIN {X 0,Y 379.102,Z 587.873,A -85,B 0,C 180,E1 -12313.302,E2 -12313.302} C_VEL
LIN {X 0,Y 377.829,Z 597.887,A -85,B 0,C 180,E1 -12314.907,E2 -12314.907} C_VEL
LIN {X 0,Y 376.972,Z 606.202,A -85,B 0,C 180,E1 -12316.525,E2 -12316.525} C_VEL
LIN {X 0,Y 375.945,Z 614.15,A -85,B 0,C 180,E1 -12318.408,E2 -12318.408} C_VEL
LIN {X 0,Y 375.318,Z 620.544,A -85,B 0,C 180,E1 -12320.299,E2 -12320.299} C_VEL
LIN {X 0,Y 374.813,Z 626.215,A -85,B 0,C 180,E1 -12322.459,E2 -12322.459} C_VEL
LIN {X 0,Y 374.699,Z 628.904,A -85,B 0,C 180,E1 -12323.767,E2 -12323.767} C_VEL
LIN {X 0,Y 374.556,Z 631.843,A -85,B 0,C 180,E1 -12325.697,E2 -12325.697} C_VEL
LIN {X 0,Y 374.414,Z 633.841,A -85,B 0,C 180,E1 -12327.85,E2 -12327.85} C_VEL
LIN {X 0,Y 374.44,Z 634.5,A -85,B 0,C 180,E1 -12330.001,E2 -12330.001} C_VEL
LIN {X 0,Y 374.414,Z 633.831,A -85,B 0,C 180,E1 -12332.153,E2 -12332.153} C_VEL
LIN {X 0,Y 374.552,Z 631.823,A -85,B 0,C 180,E1 -12334.306,E2 -12334.306} C_VEL
LIN {X 0,Y 374.678,Z 628.432,A -85,B 0,C 180,E1 -12336.463,E2 -12336.463} C_VEL
LIN {X 0,Y 375.019,Z 623.553,A -85,B 0,C 180,E1 -12338.624,E2 -12338.624} C_VEL
LIN {X 0,Y 375.479,Z 618.843,A -85,B 0,C 180,E1 -12340.244,E2 -12340.244} C_VEL
LIN {X 0,Y 376.262,Z 612.008,A -85,B 0,C 180,E1 -12342.131,E2 -12342.131} C_VEL
LIN {X 0,Y 377.062,Z 604.878,A -85,B 0,C 180,E1 -12343.749,E2 -12343.749} C_VEL
LIN {X 0,Y 378.011,Z 596.295,A -85,B 0,C 180,E1 -12345.364,E2 -12345.364} C_VEL
LIN {X 0,Y 379.327,Z 585.889,A -85,B 0,C 180,E1 -12346.968,E2 -12346.968} C_VEL
LIN {X 0,Y 380.574,Z 575.423,A -85,B 0,C 180,E1 -12348.298,E2 -12348.298} C_VEL
LIN {X 0,Y 381.89,Z 564.028,A -85,B 0,C 180,E1 -12349.486,E2 -12349.486} C_VEL
LIN {X 0,Y 383.172,Z 550.574,A -85,B 0,C 180,E1 -12350.614,E2 -12350.614} C_VEL
LIN {X 0,Y 384.244,Z 537.594,A -85,B 0,C 180,E1 -12351.459,E2 -12351.459} C_VEL
LIN {X 0,Y 385.144,Z 524.231,A -85,B 0,C 180,E1 -12352.11,E2 -12352.11} C_VEL
LIN {X 0,Y 385.838,Z 510.801,A -85,B 0,C 180,E1 -12352.561,E2 -12352.561} C_VEL
LIN {X 0,Y 386.588,Z 479.008,A -85,B 0,C 180,E1 -12353.186,E2 -12353.186} C_VEL
LIN {X 0,Y 387.875,Z 404.42,A -85,B 0,C 180,E1 -12354.584,E2 -12354.584} C_VEL
LIN {X 0,Y 383.839,Z 383.42,A -85,B 0,C 180,E1 -12355.314,E2 -12355.314} C_VEL
LIN {X 0,Y 383.618,Z 378.493,A -85,B 0,C 180,E1 -12355.793,E2 -12355.793} C_VEL
LIN {X 0,Y 380.923,Z 369.595,A -85,B 0,C 180,E1 -12357.159,E2 -12357.159} C_VEL
LIN {X 0,Y 377.404,Z 357.948,A -85,B 0,C 180,E1 -12359.341,E2 -12359.341} C_VEL
LIN {X 0,Y 375.979,Z 352.425,A -85,B 0,C 180,E1 -12360.736,E2 -12360.736} C_VEL
LIN {X 0,Y 375.967,Z 352.278,A -85,B 0,C 180,E1 -12364.112,E2 -12364.112} C_VEL
LIN {X 0,Y 375.959,Z 352.28,A -85,B 0,C 180,E1 -12366.742,E2 -12366.742} C_VEL
LIN {X 0,Y 375.993,Z 352.275,A -85,B 0,C 180,E1 -12369.971,E2 -12369.971} C_VEL
LIN {X 0,Y 375.935,Z 352.284,A -85,B 0,C 180,E1 -12373.767,E2 -12373.767} C_VEL
LIN {X 0,Y 375.938,Z 352.281,A -85,B 0,C 180,E1 -12376.811,E2 -12376.811} C_VEL
LIN {X 0,Y 375.967,Z 352.279,A -85,B 0,C 180,E1 -12380.538,E2 -12380.538} C_VEL
LIN {X 0,Y 375.993,Z 352.541,A -85,B 0,C 180,E1 -12382.318,E2 -12382.318} C_VEL
LIN {X 0,Y 378.941,Z 359.552,A -85,B 0,C 180,E1 -12384.692,E2 -12384.692} C_VEL
LIN {X 0,Y 382.121,Z 368.456,A -85,B 0,C 180,E1 -12387.213,E2 -12387.213} C_VEL
LIN {X 0,Y 384.673,Z 377.659,A -85,B 0,C 180,E1 -12389.457,E2 -12389.457} C_VEL
LIN {X 0,Y 386.067,Z 385.151,A -85,B 0,C 180,E1 -12391.069,E2 -12391.069} C_VEL
LIN {X 0,Y 384.576,Z 400.814,A -85,B 0,C 180,E1 -12393.764,E2 -12393.764} C_VEL
LIN {X 0,Y 382.802,Z 420.186,A -85,B 0,C 180,E1 -12396.995,E2 -12396.995} C_VEL
LIN {X 0,Y 386.035,Z 436.731,A -85,B 0,C 180,E1 -12397.924,E2 -12397.924} C_VEL
LIN {X 0,Y 387.355,Z 447.438,A -85,B 0,C 180,E1 -12398.409,E2 -12398.409} C_VEL
LIN {X 0,Y 384.448,Z 513.35,A -85,B 0,C 180,E1 -12400.233,E2 -12400.233} C_VEL
LIN {X 0,Y 383.578,Z 534.562,A -85,B 0,C 180,E1 -12400.848,E2 -12400.848} C_VEL
LIN {X 0,Y 382.672,Z 548.247,A -85,B 0,C 180,E1 -12401.461,E2 -12401.461} C_VEL
LIN {X 0,Y 381.718,Z 559.931,A -85,B 0,C 180,E1 -12402.176,E2 -12402.176} C_VEL
LIN {X 0,Y 380.569,Z 572.996,A -85,B 0,C 180,E1 -12403.229,E2 -12403.229} C_VEL
LIN {X 0,Y 379.407,Z 583.872,A -85,B 0,C 180,E1 -12404.334,E2 -12404.334} C_VEL
LIN {X 0,Y 378.23,Z 594.955,A -85,B 0,C 180,E1 -12405.747,E2 -12405.747} C_VEL
LIN {X 0,Y 377.263,Z 603.489,A -85,B 0,C 180,E1 -12407.083,E2 -12407.083} C_VEL
LIN {X 0,Y 376.43,Z 611.79,A -85,B 0,C 180,E1 -12408.695,E2 -12408.695} C_VEL
LIN {X 0,Y 375.723,Z 618.523,A -85,B 0,C 180,E1 -12410.308,E2 -12410.308} C_VEL
LIN {X 0,Y 375.157,Z 623.882,A -85,B 0,C 180,E1 -12411.923,E2 -12411.923} C_VEL
LIN {X 0,Y 374.802,Z 628.206,A -85,B 0,C 180,E1 -12413.631,E2 -12413.631} C_VEL
LIN {X 0,Y 374.723,Z 630.127,A -85,B 0,C 180,E1 -12414.619,E2 -12414.619} C_VEL
LIN {X 0,Y 374.591,Z 631.803,A -85,B 0,C 180,E1 -12415.696,E2 -12415.696} C_VEL
LIN {X 0,Y 374.457,Z 633.047,A -85,B 0,C 180,E1 -12416.772,E2 -12416.772} C_VEL
LIN {X 0,Y 374.436,Z 633.81,A -85,B 0,C 180,E1 -12417.849,E2 -12417.849} C_VEL
LIN {X 0,Y 374.456,Z 634.154,A -85,B 0,C 180,E1 -12418.925,E2 -12418.925} C_VEL
LIN {X 0,Y 374.444,Z 634.08,A -85,B 0,C 180,E1 -12420,E2 -12420} C_VEL
LIN {X 0,Y 374.454,Z 633.528,A -85,B 0,C 180,E1 -12421.076,E2 -12421.076} C_VEL
LIN {X 0,Y 374.419,Z 632.542,A -85,B 0,C 180,E1 -12422.152,E2 -12422.152} C_VEL
LIN {X 0,Y 374.447,Z 631.134,A -85,B 0,C 180,E1 -12423.228,E2 -12423.228} C_VEL
LIN {X 0,Y 374.595,Z 628.12,A -85,B 0,C 180,E1 -12424.843,E2 -12424.843} C_VEL
LIN {X 0,Y 374.688,Z 623.969,A -85,B 0,C 180,E1 -12426.462,E2 -12426.462} C_VEL
LIN {X 0,Y 375.002,Z 617.522,A -85,B 0,C 180,E1 -12428.352,E2 -12428.352} C_VEL
LIN {X 0,Y 375.37,Z 610.464,A -85,B 0,C 180,E1 -12429.973,E2 -12429.973} C_VEL
LIN {X 0,Y 375.95,Z 601.575,A -85,B 0,C 180,E1 -12431.593,E2 -12431.593} C_VEL
LIN {X 0,Y 376.537,Z 592.48,A -85,B 0,C 180,E1 -12432.943,E2 -12432.943} C_VEL
LIN {X 0,Y 377.262,Z 582.538,A -85,B 0,C 180,E1 -12434.146,E2 -12434.146} C_VEL
LIN {X 0,Y 378.034,Z 569.983,A -85,B 0,C 180,E1 -12435.362,E2 -12435.362} C_VEL
LIN {X 0,Y 378.739,Z 557.375,A -85,B 0,C 180,E1 -12436.3,E2 -12436.3} C_VEL
LIN {X 0,Y 379.412,Z 544.295,A -85,B 0,C 180,E1 -12437.032,E2 -12437.032} C_VEL
LIN {X 0,Y 379.945,Z 530.311,A -85,B 0,C 180,E1 -12437.562,E2 -12437.562} C_VEL
LIN {X 0,Y 381.749,Z 444.936,A -85,B 0,C 180,E1 -12439.635,E2 -12439.635} C_VEL
LIN {X 0,Y 378.693,Z 420.498,A -85,B 0,C 180,E1 -12440.394,E2 -12440.394} C_VEL
LIN {X 0,Y 380.005,Z 398.085,A -85,B 0,C 180,E1 -12444.009,E2 -12444.009} C_VEL
LIN {X 0,Y 381.299,Z 377.026,A -85,B 0,C 180,E1 -12447.438,E2 -12447.438} C_VEL
LIN {X 0,Y 379.95,Z 369.65,A -85,B 0,C 180,E1 -12448.746,E2 -12448.746} C_VEL
LIN {X 0,Y 375.982,Z 352.413,A -85,B 0,C 180,E1 -12451.934,E2 -12451.934} C_VEL
LIN {X 0,Y 375.963,Z 352.278,A -85,B 0,C 180,E1 -12455.415,E2 -12455.415} C_VEL
LIN {X 0,Y 375.978,Z 352.279,A -85,B 0,C 180,E1 -12458.27,E2 -12458.27} C_VEL
LIN {X 0,Y 375.94,Z 352.28,A -85,B 0,C 180,E1 -12461.6,E2 -12461.6} C_VEL
LIN {X 0,Y 375.932,Z 352.259,A -85,B 0,C 180,E1 -12465.268,E2 -12465.268} C_VEL
LIN {X 0,Y 375.94,Z 352.28,A -85,B 0,C 180,E1 -12468.399,E2 -12468.399} C_VEL
LIN {X 0,Y 375.981,Z 352.273,A -85,B 0,C 180,E1 -12471.729,E2 -12471.729} C_VEL
LIN {X 0,Y 375.986,Z 352.274,A -85,B 0,C 180,E1 -12475.332,E2 -12475.332} C_VEL
LIN {X 0,Y 375.969,Z 352.274,A -85,B 0,C 180,E1 -12479.167,E2 -12479.167} C_VEL
LIN {X 0,Y 376.006,Z 352.643,A -85,B 0,C 180,E1 -12479.411,E2 -12479.411} C_VEL
LIN {X 0,Y 378.515,Z 362.932,A -85,B 0,C 180,E1 -12482.041,E2 -12482.041} C_VEL
LIN {X 0,Y 380.467,Z 372.198,A -85,B 0,C 180,E1 -12484.252,E2 -12484.252} C_VEL
LIN {X 0,Y 382.895,Z 379.268,A -85,B 0,C 180,E1 -12484.61,E2 -12484.61} C_VEL
LIN {X 0,Y 387.826,Z 403.916,A -85,B 0,C 180,E1 -12485.448,E2 -12485.448} C_VEL
LIN {X 0,Y 386.4,Z 485.677,A -85,B 0,C 180,E1 -12486.979,E2 -12486.979} C_VEL
LIN {X 0,Y 385.863,Z 510.488,A -85,B 0,C 180,E1 -12487.476,E2 -12487.476} C_VEL
LIN {X 0,Y 385.084,Z 524.782,A -85,B 0,C 180,E1 -12487.957,E2 -12487.957} C_VEL
LIN {X 0,Y 384.138,Z 538.927,A -85,B 0,C 180,E1 -12488.663,E2 -12488.663} C_VEL
LIN {X 0,Y 383.131,Z 551.53,A -85,B 0,C 180,E1 -12489.505,E2 -12489.505} C_VEL
LIN {X 0,Y 381.958,Z 563.569,A -85,B 0,C 180,E1 -12490.518,E2 -12490.518} C_VEL
LIN {X 0,Y 380.599,Z 575.044,A -85,B 0,C 180,E1 -12491.703,E2 -12491.703} C_VEL
LIN {X 0,Y 379.384,Z 585.573,A -85,B 0,C 180,E1 -12493.035,E2 -12493.035} C_VEL
LIN {X 0,Y 378.08,Z 596.03,A -85,B 0,C 180,E1 -12494.638,E2 -12494.638} C_VEL
LIN {X 0,Y 377.065,Z 604.657,A -85,B 0,C 180,E1 -12496.251,E2 -12496.251} C_VEL
LIN {X 0,Y 376.107,Z 612.927,A -85,B 0,C 180,E1 -12498.137,E2 -12498.137} C_VEL
LIN {X 0,Y 375.555,Z 618.115,A -85,B 0,C 180,E1 -12499.584,E2 -12499.584} C_VEL
LIN {X 0,Y 374.671,Z 620.715,A -85,B 0,C 180,E1 -12500.383,E2 -12500.383} C_VEL
LIN {X 0,Y 371.503,Z 624.546,A -85,B 0,C 180,E1 -12501.701,E2 -12501.701} C_VEL
LIN {X 0,Y 368.877,Z 627.149,A -85,B 0,C 180,E1 -12502.793,E2 -12502.793} C_VEL
LIN {X 0,Y 367.7,Z 628.829,A -85,B 0,C 180,E1 -12503.66,E2 -12503.66} C_VEL
LIN {X 0,Y 367.574,Z 629.332,A -85,B 0,C 180,E1 -12503.957,E2 -12503.957} C_VEL
LIN {X 0,Y 367.464,Z 631.763,A -85,B 0,C 180,E1 -12505.611,E2 -12505.611} C_VEL
LIN {X 0,Y 367.319,Z 633.798,A -85,B 0,C 180,E1 -12507.806,E2 -12507.806} C_VEL
LIN {X 0,Y 367.342,Z 634.498,A -85,B 0,C 180,E1 -12509.999,E2 -12509.999} C_VEL
LIN {X 0,Y 367.318,Z 633.871,A -85,B 0,C 180,E1 -12512.192,E2 -12512.192} C_VEL
LIN {X 0,Y 367.459,Z 631.903,A -85,B 0,C 180,E1 -12514.386,E2 -12514.386} C_VEL
LIN {X 0,Y 367.624,Z 628.546,A -85,B 0,C 180,E1 -12516.585,E2 -12516.585} C_VEL
LIN {X 0,Y 367.983,Z 623.7,A -85,B 0,C 180,E1 -12518.787,E2 -12518.787} C_VEL
LIN {X 0,Y 368.597,Z 617.222,A -85,B 0,C 180,E1 -12520.99,E2 -12520.99} C_VEL
LIN {X 0,Y 369.553,Z 610.01,A -85,B 0,C 180,E1 -12522.911,E2 -12522.911} C_VEL
LIN {X 0,Y 370.48,Z 601.981,A -85,B 0,C 180,E1 -12524.654,E2 -12524.654} C_VEL
LIN {X 0,Y 371.554,Z 593.381,A -85,B 0,C 180,E1 -12526.199,E2 -12526.199} C_VEL
LIN {X 0,Y 372.967,Z 582.391,A -85,B 0,C 180,E1 -12527.829,E2 -12527.829} C_VEL
LIN {X 0,Y 374.394,Z 571.191,A -85,B 0,C 180,E1 -12529.176,E2 -12529.176} C_VEL
LIN {X 0,Y 375.755,Z 558.801,A -85,B 0,C 180,E1 -12530.385,E2 -12530.385} C_VEL
LIN {X 0,Y 376.986,Z 546.271,A -85,B 0,C 180,E1 -12531.358,E2 -12531.358} C_VEL
LIN {X 0,Y 378.009,Z 532.494,A -85,B 0,C 180,E1 -12532.187,E2 -12532.187} C_VEL
LIN {X 0,Y 378.975,Z 517.874,A -85,B 0,C 180,E1 -12532.81,E2 -12532.81} C_VEL
LIN {X 0,Y 379.569,Z 503.317,A -85,B 0,C 180,E1 -12533.204,E2 -12533.204} C_VEL
LIN {X 0,Y 381.491,Z 406.339,A -85,B 0,C 180,E1 -12535.042,E2 -12535.042} C_VEL
LIN {X 0,Y 378.899,Z 391.976,A -85,B 0,C 180,E1 -12535.52,E2 -12535.52} C_VEL
LIN {X 0,Y 376.034,Z 379.295,A -85,B 0,C 180,E1 -12535.992,E2 -12535.992} C_VEL
LIN {X 0,Y 373.275,Z 372.161,A -85,B 0,C 180,E1 -12536.391,E2 -12536.391} C_VEL
LIN {X 0,Y 370.703,Z 360.456,A -85,B 0,C 180,E1 -12539.297,E2 -12539.297} C_VEL
LIN {X 0,Y 368.974,Z 353.401,A -85,B 0,C 180,E1 -12541.178,E2 -12541.178} C_VEL
LIN {X 0,Y 368.907,Z 353.151,A -85,B 0,C 180,E1 -12542.235,E2 -12542.235} C_VEL
LIN {X 0,Y 368.925,Z 353.149,A -85,B 0,C 180,E1 -12545,E2 -12545} C_VEL
LIN {X 0,Y 368.908,Z 353.153,A -85,B 0,C 180,E1 -12548.64,E2 -12548.64} C_VEL
LIN {X 0,Y 368.946,Z 353.154,A -85,B 0,C 180,E1 -12552.02,E2 -12552.02} C_VEL
LIN {X 0,Y 368.985,Z 353.122,A -85,B 0,C 180,E1 -12555.192,E2 -12555.192} C_VEL
LIN {X 0,Y 368.934,Z 353.155,A -85,B 0,C 180,E1 -12558.185,E2 -12558.185} C_VEL
LIN {X 0,Y 368.905,Z 353.128,A -85,B 0,C 180,E1 -12561.358,E2 -12561.358} C_VEL
LIN {X 0,Y 368.928,Z 353.149,A -85,B 0,C 180,E1 -12565.145,E2 -12565.145} C_VEL
LIN {X 0,Y 368.92,Z 353.132,A -85,B 0,C 180,E1 -12569.045,E2 -12569.045} C_VEL
LIN {X 0,Y 368.977,Z 353.104,A -85,B 0,C 180,E1 -12571.564,E2 -12571.564} C_VEL
LIN {X 0,Y 368.948,Z 353.15,A -85,B 0,C 180,E1 -12575.224,E2 -12575.224} C_VEL
LIN {X 0,Y 368.927,Z 353.141,A -85,B 0,C 180,E1 -12578.973,E2 -12578.973} C_VEL
LIN {X 0,Y 368.98,Z 353.144,A -85,B 0,C 180,E1 -12582.257,E2 -12582.257} C_VEL
LIN {X 0,Y 369.027,Z 353.136,A -85,B 0,C 180,E1 -12586.227,E2 -12586.227} C_VEL
LIN {X 0,Y 369.062,Z 353.12,A -85,B 0,C 180,E1 -12590.131,E2 -12590.131} C_VEL
LIN {X 0,Y 369.177,Z 353.116,A -85,B 0,C 180,E1 -12592.342,E2 -12592.342} C_VEL
LIN {X 0,Y 369.136,Z 353.126,A -85,B 0,C 180,E1 -12594.537,E2 -12594.537} C_VEL
LIN {X 0,Y 369.309,Z 353.099,A -85,B 0,C 180,E1 -12597.819,E2 -12597.819} C_VEL
LIN {X 0,Y 369.452,Z 353.087,A -85,B 0,C 180,E1 -12600,E2 -12600} C_VEL
LIN {X 0,Y 369.309,Z 353.099,A -85,B 0,C 180,E1 -12602.181,E2 -12602.181} C_VEL
LIN {X 0,Y 369.198,Z 353.12,A -85,B 0,C 180,E1 -12606.558,E2 -12606.558} C_VEL
LIN {X 0,Y 369.128,Z 353.116,A -85,B 0,C 180,E1 -12608.761,E2 -12608.761} C_VEL
LIN {X 0,Y 369.003,Z 353.14,A -85,B 0,C 180,E1 -12612.093,E2 -12612.093} C_VEL
LIN {X 0,Y 368.988,Z 353.128,A -85,B 0,C 180,E1 -12615.465,E2 -12615.465} C_VEL
LIN {X 0,Y 368.973,Z 353.146,A -85,B 0,C 180,E1 -12618.893,E2 -12618.893} C_VEL
LIN {X 0,Y 368.923,Z 353.146,A -85,B 0,C 180,E1 -12622.396,E2 -12622.396} C_VEL
LIN {X 0,Y 368.99,Z 353.137,A -85,B 0,C 180,E1 -12625.981,E2 -12625.981} C_VEL
LIN {X 0,Y 368.895,Z 353.115,A -85,B 0,C 180,E1 -12629.692,E2 -12629.692} C_VEL
LIN {X 0,Y 368.889,Z 353.159,A -85,B 0,C 180,E1 -12633.045,E2 -12633.045} C_VEL
LIN {X 0,Y 368.909,Z 353.136,A -85,B 0,C 180,E1 -12636.198,E2 -12636.198} C_VEL
LIN {X 0,Y 368.9,Z 353.132,A -85,B 0,C 180,E1 -12638.954,E2 -12638.954} C_VEL
LIN {X 0,Y 368.944,Z 353.154,A -85,B 0,C 180,E1 -12642.023,E2 -12642.023} C_VEL
LIN {X 0,Y 368.984,Z 353.124,A -85,B 0,C 180,E1 -12645.194,E2 -12645.194} C_VEL
LIN {X 0,Y 368.939,Z 353.152,A -85,B 0,C 180,E1 -12648.188,E2 -12648.188} C_VEL
LIN {X 0,Y 368.908,Z 353.152,A -85,B 0,C 180,E1 -12651.36,E2 -12651.36} C_VEL
LIN {X 0,Y 368.931,Z 353.15,A -85,B 0,C 180,E1 -12655.148,E2 -12655.148} C_VEL
LIN {X 0,Y 368.949,Z 353.295,A -85,B 0,C 180,E1 -12658.82,E2 -12658.82} C_VEL
LIN {X 0,Y 371.652,Z 364.514,A -85,B 0,C 180,E1 -12661.789,E2 -12661.789} C_VEL
LIN {X 0,Y 373.316,Z 372.35,A -85,B 0,C 180,E1 -12663.676,E2 -12663.676} C_VEL
LIN {X 0,Y 376.605,Z 380.966,A -85,B 0,C 180,E1 -12664.13,E2 -12664.13} C_VEL
LIN {X 0,Y 381.439,Z 405.172,A -85,B 0,C 180,E1 -12664.976,E2 -12664.976} C_VEL
LIN {X 0,Y 379.78,Z 492.274,A -85,B 0,C 180,E1 -12666.629,E2 -12666.629} C_VEL
LIN {X 0,Y 379.246,Z 512.408,A -85,B 0,C 180,E1 -12667.063,E2 -12667.063} C_VEL
LIN {X 0,Y 378.451,Z 526.818,A -85,B 0,C 180,E1 -12667.589,E2 -12667.589} C_VEL
LIN {X 0,Y 377.483,Z 540.12,A -85,B 0,C 180,E1 -12668.287,E2 -12668.287} C_VEL
LIN {X 0,Y 376.33,Z 553.498,A -85,B 0,C 180,E1 -12669.219,E2 -12669.219} C_VEL
LIN {X 0,Y 375.057,Z 565.597,A -85,B 0,C 180,E1 -12670.29,E2 -12670.29} C_VEL
LIN {X 0,Y 373.552,Z 577.799,A -85,B 0,C 180,E1 -12671.633,E2 -12671.633} C_VEL
LIN {X 0,Y 372.292,Z 587.876,A -85,B 0,C 180,E1 -12672.988,E2 -12672.988} C_VEL
LIN {X 0,Y 370.947,Z 597.889,A -85,B 0,C 180,E1 -12674.62,E2 -12674.62} C_VEL
LIN {X 0,Y 369.994,Z 606.204,A -85,B 0,C 180,E1 -12676.266,E2 -12676.266} C_VEL
LIN {X 0,Y 368.967,Z 614.151,A -85,B 0,C 180,E1 -12678.186,E2 -12678.186} C_VEL
LIN {X 0,Y 368.275,Z 620.545,A -85,B 0,C 180,E1 -12680.112,E2 -12680.112} C_VEL
LIN {X 0,Y 367.737,Z 626.216,A -85,B 0,C 180,E1 -12682.313,E2 -12682.313} C_VEL
LIN {X 0,Y 367.521,Z 630.33,A -85,B 0,C 180,E1 -12684.515,E2 -12684.515} C_VEL
LIN {X 0,Y 367.358,Z 633.012,A -85,B 0,C 180,E1 -12686.711,E2 -12686.711} C_VEL
LIN {X 0,Y 367.348,Z 634.337,A -85,B 0,C 180,E1 -12688.905,E2 -12688.905} C_VEL
LIN {X 0,Y 367.348,Z 634.332,A -85,B 0,C 180,E1 -12691.098,E2 -12691.098} C_VEL
LIN {X 0,Y 367.358,Z 632.996,A -85,B 0,C 180,E1 -12693.292,E2 -12693.292} C_VEL
LIN {X 0,Y 367.498,Z 630.305,A -85,B 0,C 180,E1 -12695.488,E2 -12695.488} C_VEL
LIN {X 0,Y 367.738,Z 626.186,A -85,B 0,C 180,E1 -12697.689,E2 -12697.689} C_VEL
LIN {X 0,Y 368.277,Z 620.509,A -85,B 0,C 180,E1 -12699.891,E2 -12699.891} C_VEL
LIN {X 0,Y 368.968,Z 614.102,A -85,B 0,C 180,E1 -12701.817,E2 -12701.817} C_VEL
LIN {X 0,Y 369.997,Z 606.144,A -85,B 0,C 180,E1 -12703.736,E2 -12703.736} C_VEL
LIN {X 0,Y 370.954,Z 597.815,A -85,B 0,C 180,E1 -12705.382,E2 -12705.382} C_VEL
LIN {X 0,Y 372.283,Z 587.786,A -85,B 0,C 180,E1 -12707.016,E2 -12707.016} C_VEL
LIN {X 0,Y 373.681,Z 576.593,A -85,B 0,C 180,E1 -12708.506,E2 -12708.506} C_VEL
LIN {X 0,Y 375.174,Z 564.024,A -85,B 0,C 180,E1 -12709.849,E2 -12709.849} C_VEL
LIN {X 0,Y 376.477,Z 551.2,A -85,B 0,C 180,E1 -12710.947,E2 -12710.947} C_VEL
LIN {X 0,Y 377.635,Z 537.588,A -85,B 0,C 180,E1 -12711.853,E2 -12711.853} C_VEL
LIN {X 0,Y 378.588,Z 524.222,A -85,B 0,C 180,E1 -12712.513,E2 -12712.513} C_VEL
LIN {X 0,Y 379.313,Z 510.789,A -85,B 0,C 180,E1 -12712.971,E2 -12712.971} C_VEL
LIN {X 0,Y 380.093,Z 478.988,A -85,B 0,C 180,E1 -12713.606,E2 -12713.606} C_VEL
LIN {X 0,Y 381.436,Z 405.55,A -85,B 0,C 180,E1 -12715.004,E2 -12715.004} C_VEL
LIN {X 0,Y 378.329,Z 389.189,A -85,B 0,C 180,E1 -12715.578,E2 -12715.578} C_VEL
LIN {X 0,Y 378.39,Z 383.101,A -85,B 0,C 180,E1 -12716.142,E2 -12716.142} C_VEL
LIN {X 0,Y 376.498,Z 375.752,A -85,B 0,C 180,E1 -12717.236,E2 -12717.236} C_VEL
LIN {X 0,Y 373.162,Z 364.587,A -85,B 0,C 180,E1 -12719.32,E2 -12719.32} C_VEL
LIN {X 0,Y 371.405,Z 358.26,A -85,B 0,C 180,E1 -12720.726,E2 -12720.726} C_VEL
LIN {X 0,Y 369.071,Z 354.015,A -85,B 0,C 180,E1 -12722.222,E2 -12722.222} C_VEL
LIN {X 0,Y 368.937,Z 353.273,A -85,B 0,C 180,E1 -12722.637,E2 -12722.637} C_VEL
LIN {X 0,Y 368.923,Z 353.154,A -85,B 0,C 180,E1 -12726.197,E2 -12726.197} C_VEL
LIN {X 0,Y 368.909,Z 353.157,A -85,B 0,C 180,E1 -12728.954,E2 -12728.954} C_VEL
LIN {X 0,Y 368.886,Z 353.162,A -85,B 0,C 180,E1 -12732.01,E2 -12732.01} C_VEL
LIN {X 0,Y 368.884,Z 353.16,A -85,B 0,C 180,E1 -12735.176,E2 -12735.176} C_VEL
LIN {X 0,Y 368.887,Z 353.159,A -85,B 0,C 180,E1 -12738.178,E2 -12738.178} C_VEL
LIN {X 0,Y 368.969,Z 353.419,A -85,B 0,C 180,E1 -12740.571,E2 -12740.571} C_VEL
LIN {X 0,Y 371.196,Z 358.664,A -85,B 0,C 180,E1 -12742.709,E2 -12742.709} C_VEL
LIN {X 0,Y 373.829,Z 364.987,A -85,B 0,C 180,E1 -12744.866,E2 -12744.866} C_VEL
LIN {X 0,Y 376.492,Z 372.865,A -85,B 0,C 180,E1 -12747.144,E2 -12747.144} C_VEL
LIN {X 0,Y 378.718,Z 381.236,A -85,B 0,C 180,E1 -12749.248,E2 -12749.248} C_VEL
LIN {X 0,Y 379.875,Z 388.756,A -85,B 0,C 180,E1 -12750.903,E2 -12750.903} C_VEL
LIN {X 0,Y 377.497,Z 410.283,A -85,B 0,C 180,E1 -12754.647,E2 -12754.647} C_VEL
LIN {X 0,Y 376.58,Z 420.093,A -85,B 0,C 180,E1 -12756.3,E2 -12756.3} C_VEL
LIN {X 0,Y 379.875,Z 436.734,A -85,B 0,C 180,E1 -12757.298,E2 -12757.298} C_VEL
LIN {X 0,Y 381.36,Z 448.852,A -85,B 0,C 180,E1 -12757.88,E2 -12757.88} C_VEL
LIN {X 0,Y 378.075,Z 515.539,A -85,B 0,C 180,E1 -12759.779,E2 -12759.779} C_VEL
LIN {X 0,Y 377.25,Z 534.904,A -85,B 0,C 180,E1 -12760.372,E2 -12760.372} C_VEL
LIN {X 0,Y 376.29,Z 548.378,A -85,B 0,C 180,E1 -12760.993,E2 -12760.993} C_VEL
LIN {X 0,Y 375.263,Z 559.959,A -85,B 0,C 180,E1 -12761.718,E2 -12761.718} C_VEL
LIN {X 0,Y 374.042,Z 572.96,A -85,B 0,C 180,E1 -12762.787,E2 -12762.787} C_VEL
LIN {X 0,Y 372.873,Z 583.517,A -85,B 0,C 180,E1 -12763.877,E2 -12763.877} C_VEL
LIN {X 0,Y 371.647,Z 593.921,A -85,B 0,C 180,E1 -12765.209,E2 -12765.209} C_VEL
LIN {X 0,Y 370.643,Z 602.606,A -85,B 0,C 180,E1 -12766.569,E2 -12766.569} C_VEL
LIN {X 0,Y 369.825,Z 609.813,A -85,B 0,C 180,E1 -12767.934,E2 -12767.934} C_VEL
LIN {X 0,Y 368.937,Z 616.921,A -85,B 0,C 180,E1 -12769.574,E2 -12769.574} C_VEL
LIN {X 0,Y 368.301,Z 622.585,A -85,B 0,C 180,E1 -12771.219,E2 -12771.219} C_VEL
LIN {X 0,Y 367.859,Z 627.016,A -85,B 0,C 180,E1 -12772.866,E2 -12772.866} C_VEL
LIN {X 0,Y 367.652,Z 630.32,A -85,B 0,C 180,E1 -12774.515,E2 -12774.515} C_VEL
LIN {X 0,Y 367.527,Z 631.958,A -85,B 0,C 180,E1 -12775.613,E2 -12775.613} C_VEL
LIN {X 0,Y 367.378,Z 633.132,A -85,B 0,C 180,E1 -12776.71,E2 -12776.71} C_VEL
LIN {X 0,Y 367.339,Z 633.853,A -85,B 0,C 180,E1 -12777.807,E2 -12777.807} C_VEL
LIN {X 0,Y 367.355,Z 634.159,A -85,B 0,C 180,E1 -12778.904,E2 -12778.904} C_VEL
LIN {X 0,Y 367.344,Z 634.022,A -85,B 0,C 180,E1 -12780,E2 -12780} C_VEL
LIN {X 0,Y 367.353,Z 633.414,A -85,B 0,C 180,E1 -12781.096,E2 -12781.096} C_VEL
LIN {X 0,Y 367.323,Z 632.388,A -85,B 0,C 180,E1 -12782.193,E2 -12782.193} C_VEL
LIN {X 0,Y 367.368,Z 630.917,A -85,B 0,C 180,E1 -12783.29,E2 -12783.29} C_VEL
LIN {X 0,Y 367.51,Z 627.8,A -85,B 0,C 180,E1 -12784.937,E2 -12784.937} C_VEL
LIN {X 0,Y 367.631,Z 623.535,A -85,B 0,C 180,E1 -12786.587,E2 -12786.587} C_VEL
LIN {X 0,Y 367.958,Z 616.973,A -85,B 0,C 180,E1 -12788.513,E2 -12788.513} C_VEL
LIN {X 0,Y 368.344,Z 609.736,A -85,B 0,C 180,E1 -12790.165,E2 -12790.165} C_VEL
LIN {X 0,Y 368.948,Z 600.689,A -85,B 0,C 180,E1 -12791.816,E2 -12791.816} C_VEL
LIN {X 0,Y 369.549,Z 591.378,A -85,B 0,C 180,E1 -12793.192,E2 -12793.192} C_VEL
LIN {X 0,Y 370.23,Z 582.376,A -85,B 0,C 180,E1 -12794.287,E2 -12794.287} C_VEL
LIN {X 0,Y 371.028,Z 569.872,A -85,B 0,C 180,E1 -12795.519,E2 -12795.519} C_VEL
LIN {X 0,Y 371.744,Z 557.248,A -85,B 0,C 180,E1 -12796.474,E2 -12796.474} C_VEL
LIN {X 0,Y 372.435,Z 544.174,A -85,B 0,C 180,E1 -12797.219,E2 -12797.219} C_VEL
LIN {X 0,Y 372.981,Z 530.25,A -85,B 0,C 180,E1 -12797.759,E2 -12797.759} C_VEL
LIN {X 0,Y 374.851,Z 445.493,A -85,B 0,C 180,E1 -12799.875,E2 -12799.875} C_VEL
LIN {X 0,Y 371.778,Z 420.489,A -85,B 0,C 180,E1 -12800.671,E2 -12800.671} C_VEL
LIN {X 0,Y 373.056,Z 398.937,A -85,B 0,C 180,E1 -12804.189,E2 -12804.189} C_VEL
LIN {X 0,Y 374.389,Z 378.374,A -85,B 0,C 180,E1 -12807.582,E2 -12807.582} C_VEL
LIN {X 0,Y 372.815,Z 370.241,A -85,B 0,C 180,E1 -12809.04,E2 -12809.04} C_VEL
LIN {X 0,Y 368.951,Z 353.325,A -85,B 0,C 180,E1 -12812.2,E2 -12812.2} C_VEL
LIN {X 0,Y 368.935,Z 353.154,A -85,B 0,C 180,E1 -12815.001,E2 -12815.001} C_VEL
LIN {X 0,Y 368.912,Z 353.158,A -85,B 0,C 180,E1 -12818.639,E2 -12818.639} C_VEL
LIN {X 0,Y 368.887,Z 353.162,A -85,B 0,C 180,E1 -12822.009,E2 -12822.009} C_VEL
LIN {X 0,Y 368.885,Z 353.136,A -85,B 0,C 180,E1 -12825.175,E2 -12825.175} C_VEL
LIN {X 0,Y 368.889,Z 353.161,A -85,B 0,C 180,E1 -12828.177,E2 -12828.177} C_VEL
LIN {X 0,Y 368.915,Z 353.15,A -85,B 0,C 180,E1 -12831.359,E2 -12831.359} C_VEL
LIN {X 0,Y 368.942,Z 353.148,A -85,B 0,C 180,E1 -12835.146,E2 -12835.146} C_VEL
LIN {X 0,Y 368.949,Z 353.33,A -85,B 0,C 180,E1 -12838.904,E2 -12838.904} C_VEL
LIN {X 0,Y 371.608,Z 364.242,A -85,B 0,C 180,E1 -12841.782,E2 -12841.782} C_VEL
LIN {X 0,Y 373.257,Z 372.172,A -85,B 0,C 180,E1 -12843.712,E2 -12843.712} C_VEL
LIN {X 0,Y 376.492,Z 380.554,A -85,B 0,C 180,E1 -12844.172,E2 -12844.172} C_VEL
LIN {X 0,Y 381.469,Z 405.832,A -85,B 0,C 180,E1 -12845.049,E2 -12845.049} C_VEL
LIN {X 0,Y 379.359,Z 509.355,A -85,B 0,C 180,E1 -12847.032,E2 -12847.032} C_VEL
LIN {X 0,Y 378.58,Z 524.031,A -85,B 0,C 180,E1 -12847.522,E2 -12847.522} C_VEL
LIN {X 0,Y 377.705,Z 536.88,A -85,B 0,C 180,E1 -12848.151,E2 -12848.151} C_VEL
LIN {X 0,Y 376.608,Z 550.015,A -85,B 0,C 180,E1 -12849.01,E2 -12849.01} C_VEL
LIN {X 0,Y 375.38,Z 562.149,A -85,B 0,C 180,E1 -12850.019,E2 -12850.019} C_VEL
LIN {X 0,Y 374.044,Z 573.875,A -85,B 0,C 180,E1 -12851.229,E2 -12851.229} C_VEL
LIN {X 0,Y 372.785,Z 583.627,A -85,B 0,C 180,E1 -12852.442,E2 -12852.442} C_VEL
LIN {X 0,Y 371.395,Z 594.406,A -85,B 0,C 180,E1 -12854.073,E2 -12854.073} C_VEL
LIN {X 0,Y 370.274,Z 603.306,A -85,B 0,C 180,E1 -12855.714,E2 -12855.714} C_VEL
LIN {X 0,Y 369.434,Z 610.711,A -85,B 0,C 180,E1 -12857.362,E2 -12857.362} C_VEL
LIN {X 0,Y 368.646,Z 616.886,A -85,B 0,C 180,E1 -12859.008,E2 -12859.008} C_VEL
LIN {X 0,Y 367.99,Z 623.436,A -85,B 0,C 180,E1 -12861.21,E2 -12861.21} C_VEL
LIN {X 0,Y 367.592,Z 628.344,A -85,B 0,C 180,E1 -12863.412,E2 -12863.412} C_VEL
LIN {X 0,Y 367.574,Z 629.332,A -85,B 0,C 180,E1 -12863.957,E2 -12863.957} C_VEL
LIN {X 0,Y 366.791,Z 630.766,A -85,B 0,C 180,E1 -12864.846,E2 -12864.846} C_VEL
LIN {X 0,Y 363.786,Z 632.57,A -85,B 0,C 180,E1 -12866.301,E2 -12866.301} C_VEL
LIN {X 0,Y 361.321,Z 633.597,A -85,B 0,C 180,E1 -12867.489,E2 -12867.489} C_VEL
LIN {X 0,Y 360.301,Z 634.114,A -85,B 0,C 180,E1 -12868.414,E2 -12868.414} C_VEL
LIN {X 0,Y 360.236,Z 634.243,A -85,B 0,C 180,E1 -12868.727,E2 -12868.727} C_VEL
LIN {X 0,Y 360.242,Z 634.498,A -85,B 0,C 180,E1 -12869.999,E2 -12869.999} C_VEL
LIN {X 0,Y 360.225,Z 633.87,A -85,B 0,C 180,E1 -12872.235,E2 -12872.235} C_VEL
LIN {X 0,Y 360.37,Z 631.903,A -85,B 0,C 180,E1 -12874.473,E2 -12874.473} C_VEL
LIN {X 0,Y 360.563,Z 628.545,A -85,B 0,C 180,E1 -12876.715,E2 -12876.715} C_VEL
LIN {X 0,Y 360.925,Z 623.699,A -85,B 0,C 180,E1 -12878.96,E2 -12878.96} C_VEL
LIN {X 0,Y 361.429,Z 619.028,A -85,B 0,C 180,E1 -12880.644,E2 -12880.644} C_VEL
LIN {X 0,Y 362.321,Z 612.24,A -85,B 0,C 180,E1 -12882.603,E2 -12882.603} C_VEL
LIN {X 0,Y 363.337,Z 603.804,A -85,B 0,C 180,E1 -12884.562,E2 -12884.562} C_VEL
LIN {X 0,Y 364.48,Z 595.004,A -85,B 0,C 180,E1 -12886.234,E2 -12886.234} C_VEL
LIN {X 0,Y 365.916,Z 584.341,A -85,B 0,C 180,E1 -12887.895,E2 -12887.895} C_VEL
LIN {X 0,Y 367.375,Z 573.56,A -85,B 0,C 180,E1 -12889.267,E2 -12889.267} C_VEL
LIN {X 0,Y 368.744,Z 561.768,A -85,B 0,C 180,E1 -12890.499,E2 -12890.499} C_VEL
LIN {X 0,Y 370.111,Z 549.241,A -85,B 0,C 180,E1 -12891.544,E2 -12891.544} C_VEL
LIN {X 0,Y 371.202,Z 536.255,A -85,B 0,C 180,E1 -12892.396,E2 -12892.396} C_VEL
LIN {X 0,Y 372.18,Z 522.406,A -85,B 0,C 180,E1 -12893.067,E2 -12893.067} C_VEL
LIN {X 0,Y 372.934,Z 507.808,A -85,B 0,C 180,E1 -12893.532,E2 -12893.532} C_VEL
LIN {X 0,Y 375.069,Z 407.13,A -85,B 0,C 180,E1 -12895.484,E2 -12895.484} C_VEL
LIN {X 0,Y 370.898,Z 385.671,A -85,B 0,C 180,E1 -12896.244,E2 -12896.244} C_VEL
LIN {X 0,Y 369.634,Z 381.126,A -85,B 0,C 180,E1 -12896.437,E2 -12896.437} C_VEL
LIN {X 0,Y 366.08,Z 372.286,A -85,B 0,C 180,E1 -12896.937,E2 -12896.937} C_VEL
LIN {X 0,Y 363.735,Z 361.737,A -85,B 0,C 180,E1 -12899.602,E2 -12899.602} C_VEL
LIN {X 0,Y 361.915,Z 354.135,A -85,B 0,C 180,E1 -12901.702,E2 -12901.702} C_VEL
LIN {X 0,Y 361.864,Z 354.023,A -85,B 0,C 180,E1 -12905.635,E2 -12905.635} C_VEL
LIN {X 0,Y 361.87,Z 354.023,A -85,B 0,C 180,E1 -12909.026,E2 -12909.026} C_VEL
LIN {X 0,Y 361.886,Z 354.032,A -85,B 0,C 180,E1 -12912.44,E2 -12912.44} C_VEL
LIN {X 0,Y 361.923,Z 354.004,A -85,B 0,C 180,E1 -12915.927,E2 -12915.927} C_VEL
LIN {X 0,Y 361.898,Z 354.03,A -85,B 0,C 180,E1 -12919.23,E2 -12919.23} C_VEL
LIN {X 0,Y 361.861,Z 354.003,A -85,B 0,C 180,E1 -12922.981,E2 -12922.981} C_VEL
LIN {X 0,Y 361.852,Z 354.035,A -85,B 0,C 180,E1 -12926.629,E2 -12926.629} C_VEL
LIN {X 0,Y 361.867,Z 353.998,A -85,B 0,C 180,E1 -12929.671,E2 -12929.671} C_VEL
LIN {X 0,Y 361.945,Z 354.005,A -85,B 0,C 180,E1 -12933.474,E2 -12933.474} C_VEL
LIN {X 0,Y 361.881,Z 354.031,A -85,B 0,C 180,E1 -12937.144,E2 -12937.144} C_VEL
LIN {X 0,Y 361.911,Z 354.024,A -85,B 0,C 180,E1 -12940.723,E2 -12940.723} C_VEL
LIN {X 0,Y 361.936,Z 354.008,A -85,B 0,C 180,E1 -12944.226,E2 -12944.226} C_VEL
LIN {X 0,Y 361.99,Z 354.013,A -85,B 0,C 180,E1 -12946.527,E2 -12946.527} C_VEL
LIN {X 0,Y 362.026,Z 353.997,A -85,B 0,C 180,E1 -12949.938,E2 -12949.938} C_VEL
LIN {X 0,Y 362.14,Z 353.993,A -85,B 0,C 180,E1 -12952.192,E2 -12952.192} C_VEL
LIN {X 0,Y 362.11,Z 354.001,A -85,B 0,C 180,E1 -12954.431,E2 -12954.431} C_VEL
LIN {X 0,Y 362.273,Z 353.975,A -85,B 0,C 180,E1 -12957.776,E2 -12957.776} C_VEL
LIN {X 0,Y 362.421,Z 353.963,A -85,B 0,C 180,E1 -12960,E2 -12960} C_VEL
LIN {X 0,Y 362.273,Z 353.975,A -85,B 0,C 180,E1 -12962.224,E2 -12962.224} C_VEL
LIN {X 0,Y 362.162,Z 353.998,A -85,B 0,C 180,E1 -12966.686,E2 -12966.686} C_VEL
LIN {X 0,Y 362.065,Z 353.993,A -85,B 0,C 180,E1 -12968.933,E2 -12968.933} C_VEL
LIN {X 0,Y 361.957,Z 354.019,A -85,B 0,C 180,E1 -12972.332,E2 -12972.332} C_VEL
LIN {X 0,Y 361.952,Z 354.01,A -85,B 0,C 180,E1 -12974.621,E2 -12974.621} C_VEL
LIN {X 0,Y 361.949,Z 354.019,A -85,B 0,C 180,E1 -12978.1,E2 -12978.1} C_VEL
LIN {X 0,Y 361.882,Z 354.018,A -85,B 0,C 180,E1 -12981.653,E2 -12981.653} C_VEL
LIN {X 0,Y 361.918,Z 354.021,A -85,B 0,C 180,E1 -12985.291,E2 -12985.291} C_VEL
LIN {X 0,Y 361.898,Z 353.993,A -85,B 0,C 180,E1 -12987.78,E2 -12987.78} C_VEL
LIN {X 0,Y 361.828,Z 354.027,A -85,B 0,C 180,E1 -12991.63,E2 -12991.63} C_VEL
LIN {X 0,Y 361.866,Z 354.027,A -85,B 0,C 180,E1 -12995.346,E2 -12995.346} C_VEL
LIN {X 0,Y 361.866,Z 354.008,A -85,B 0,C 180,E1 -12999.029,E2 -12999.029} C_VEL
LIN {X 0,Y 361.885,Z 354.028,A -85,B 0,C 180,E1 -13002.443,E2 -13002.443} C_VEL
LIN {X 0,Y 361.923,Z 354.01,A -85,B 0,C 180,E1 -13005.929,E2 -13005.929} C_VEL
LIN {X 0,Y 361.9,Z 354.019,A -85,B 0,C 180,E1 -13009.233,E2 -13009.233} C_VEL
LIN {X 0,Y 361.868,Z 354.031,A -85,B 0,C 180,E1 -13012.984,E2 -13012.984} C_VEL
LIN {X 0,Y 361.859,Z 354.029,A -85,B 0,C 180,E1 -13016.631,E2 -13016.631} C_VEL
LIN {X 0,Y 361.942,Z 354.2,A -85,B 0,C 180,E1 -13018.383,E2 -13018.383} C_VEL
LIN {X 0,Y 364.683,Z 365.764,A -85,B 0,C 180,E1 -13021.5,E2 -13021.5} C_VEL
LIN {X 0,Y 366.143,Z 372.385,A -85,B 0,C 180,E1 -13023.121,E2 -13023.121} C_VEL
LIN {X 0,Y 370.546,Z 383.809,A -85,B 0,C 180,E1 -13023.735,E2 -13023.735} C_VEL
LIN {X 0,Y 375.058,Z 406.59,A -85,B 0,C 180,E1 -13024.549,E2 -13024.549} C_VEL
LIN {X 0,Y 372.955,Z 507.473,A -85,B 0,C 180,E1 -13026.507,E2 -13026.507} C_VEL
LIN {X 0,Y 372.195,Z 522.216,A -85,B 0,C 180,E1 -13026.971,E2 -13026.971} C_VEL
LIN {X 0,Y 371.225,Z 535.554,A -85,B 0,C 180,E1 -13027.606,E2 -13027.606} C_VEL
LIN {X 0,Y 370.096,Z 549.385,A -85,B 0,C 180,E1 -13028.512,E2 -13028.512} C_VEL
LIN {X 0,Y 368.885,Z 561.328,A -85,B 0,C 180,E1 -13029.509,E2 -13029.509} C_VEL
LIN {X 0,Y 367.403,Z 573.196,A -85,B 0,C 180,E1 -13030.735,E2 -13030.735} C_VEL
LIN {X 0,Y 365.977,Z 584.037,A -85,B 0,C 180,E1 -13032.108,E2 -13032.108} C_VEL
LIN {X 0,Y 364.489,Z 594.75,A -85,B 0,C 180,E1 -13033.766,E2 -13033.766} C_VEL
LIN {X 0,Y 363.329,Z 603.591,A -85,B 0,C 180,E1 -13035.437,E2 -13035.437} C_VEL
LIN {X 0,Y 362.466,Z 610.948,A -85,B 0,C 180,E1 -13037.118,E2 -13037.118} C_VEL
LIN {X 0,Y 361.602,Z 617.077,A -85,B 0,C 180,E1 -13038.794,E2 -13038.794} C_VEL
LIN {X 0,Y 360.925,Z 623.585,A -85,B 0,C 180,E1 -13041.04,E2 -13041.04} C_VEL
LIN {X 0,Y 360.57,Z 628.46,A -85,B 0,C 180,E1 -13043.285,E2 -13043.285} C_VEL
LIN {X 0,Y 360.377,Z 631.844,A -85,B 0,C 180,E1 -13045.527,E2 -13045.527} C_VEL
LIN {X 0,Y 360.225,Z 633.842,A -85,B 0,C 180,E1 -13047.765,E2 -13047.765} C_VEL
LIN {X 0,Y 360.241,Z 634.5,A -85,B 0,C 180,E1 -13050.001,E2 -13050.001} C_VEL
LIN {X 0,Y 360.225,Z 633.831,A -85,B 0,C 180,E1 -13052.238,E2 -13052.238} C_VEL
LIN {X 0,Y 360.371,Z 631.822,A -85,B 0,C 180,E1 -13054.475,E2 -13054.475} C_VEL
LIN {X 0,Y 360.512,Z 628.43,A -85,B 0,C 180,E1 -13056.718,E2 -13056.718} C_VEL
LIN {X 0,Y 360.927,Z 623.551,A -85,B 0,C 180,E1 -13058.963,E2 -13058.963} C_VEL
LIN {X 0,Y 361.44,Z 618.84,A -85,B 0,C 180,E1 -13060.646,E2 -13060.646} C_VEL
LIN {X 0,Y 362.337,Z 612.005,A -85,B 0,C 180,E1 -13062.605,E2 -13062.605} C_VEL
LIN {X 0,Y 363.334,Z 603.521,A -85,B 0,C 180,E1 -13064.565,E2 -13064.565} C_VEL
LIN {X 0,Y 364.519,Z 594.664,A -85,B 0,C 180,E1 -13066.235,E2 -13066.235} C_VEL
LIN {X 0,Y 365.936,Z 583.934,A -85,B 0,C 180,E1 -13067.897,E2 -13067.897} C_VEL
LIN {X 0,Y 367.42,Z 573.069,A -85,B 0,C 180,E1 -13069.267,E2 -13069.267} C_VEL
LIN {X 0,Y 368.832,Z 561.169,A -85,B 0,C 180,E1 -13070.497,E2 -13070.497} C_VEL
LIN {X 0,Y 370.148,Z 548.188,A -85,B 0,C 180,E1 -13071.571,E2 -13071.571} C_VEL
LIN {X 0,Y 371.327,Z 534.012,A -85,B 0,C 180,E1 -13072.464,E2 -13072.464} C_VEL
LIN {X 0,Y 372.264,Z 520.001,A -85,B 0,C 180,E1 -13073.101,E2 -13073.101} C_VEL
LIN {X 0,Y 372.943,Z 505.296,A -85,B 0,C 180,E1 -13073.534,E2 -13073.534} C_VEL
LIN {X 0,Y 375.032,Z 406.601,A -85,B 0,C 180,E1 -13075.439,E2 -13075.439} C_VEL
LIN {X 0,Y 372.8,Z 394.643,A -85,B 0,C 180,E1 -13075.876,E2 -13075.876} C_VEL
LIN {X 0,Y 373.02,Z 386.273,A -85,B 0,C 180,E1 -13076.677,E2 -13076.677} C_VEL
LIN {X 0,Y 370.944,Z 378.191,A -85,B 0,C 180,E1 -13077.966,E2 -13077.966} C_VEL
LIN {X 0,Y 367.875,Z 366.765,A -85,B 0,C 180,E1 -13080.226,E2 -13080.226} C_VEL
LIN {X 0,Y 366.673,Z 363.065,A -85,B 0,C 180,E1 -13081.166,E2 -13081.166} C_VEL
LIN {X 0,Y 364.462,Z 358.764,A -85,B 0,C 180,E1 -13082.68,E2 -13082.68} C_VEL
LIN {X 0,Y 362.309,Z 355.766,A -85,B 0,C 180,E1 -13084.233,E2 -13084.233} C_VEL
LIN {X 0,Y 361.924,Z 354.203,A -85,B 0,C 180,E1 -13085.048,E2 -13085.048} C_VEL
LIN {X 0,Y 361.874,Z 354.035,A -85,B 0,C 180,E1 -13088.425,E2 -13088.425} C_VEL
LIN {X 0,Y 361.832,Z 354.036,A -85,B 0,C 180,E1 -13091.331,E2 -13091.331} C_VEL
LIN {X 0,Y 361.822,Z 354.039,A -85,B 0,C 180,E1 -13094.369,E2 -13094.369} C_VEL
LIN {X 0,Y 361.875,Z 354.234,A -85,B 0,C 180,E1 -13098.118,E2 -13098.118} C_VEL
LIN {X 0,Y 363.106,Z 357.228,A -85,B 0,C 180,E1 -13099.815,E2 -13099.815} C_VEL
LIN {X 0,Y 363.94,Z 358.647,A -85,B 0,C 180,E1 -13100.575,E2 -13100.575} C_VEL
LIN {X 0,Y 366.345,Z 364.197,A -85,B 0,C 180,E1 -13102.893,E2 -13102.893} C_VEL
LIN {X 0,Y 368.83,Z 370.68,A -85,B 0,C 180,E1 -13105.135,E2 -13105.135} C_VEL
LIN {X 0,Y 370.979,Z 377.661,A -85,B 0,C 180,E1 -13107.177,E2 -13107.177} C_VEL
LIN {X 0,Y 372.857,Z 385.168,A -85,B 0,C 180,E1 -13109.102,E2 -13109.102} C_VEL
LIN {X 0,Y 373.788,Z 391.018,A -85,B 0,C 180,E1 -13110.437,E2 -13110.437} C_VEL
LIN {X 0,Y 371.686,Z 408.816,A -85,B 0,C 180,E1 -13113.618,E2 -13113.618} C_VEL
LIN {X 0,Y 370.504,Z 420.265,A -85,B 0,C 180,E1 -13115.577,E2 -13115.577} C_VEL
LIN {X 0,Y 373.672,Z 436.113,A -85,B 0,C 180,E1 -13116.594,E2 -13116.594} C_VEL
LIN {X 0,Y 375.43,Z 449.121,A -85,B 0,C 180,E1 -13117.276,E2 -13117.276} C_VEL
LIN {X 0,Y 372.065,Z 513.504,A -85,B 0,C 180,E1 -13119.185,E2 -13119.185} C_VEL
LIN {X 0,Y 371.006,Z 534.797,A -85,B 0,C 180,E1 -13119.847,E2 -13119.847} C_VEL
LIN {X 0,Y 370.028,Z 547.559,A -85,B 0,C 180,E1 -13120.442,E2 -13120.442} C_VEL
LIN {X 0,Y 368.858,Z 560.177,A -85,B 0,C 180,E1 -13121.245,E2 -13121.245} C_VEL
LIN {X 0,Y 367.553,Z 573.077,A -85,B 0,C 180,E1 -13122.329,E2 -13122.329} C_VEL
LIN {X 0,Y 366.136,Z 584.7,A -85,B 0,C 180,E1 -13123.571,E2 -13123.571} C_VEL
LIN {X 0,Y 364.854,Z 594.903,A -85,B 0,C 180,E1 -13124.927,E2 -13124.927} C_VEL
LIN {X 0,Y 363.8,Z 603.403,A -85,B 0,C 180,E1 -13126.311,E2 -13126.311} C_VEL
LIN {X 0,Y 362.734,Z 611.709,A -85,B 0,C 180,E1 -13127.978,E2 -13127.978} C_VEL
LIN {X 0,Y 361.879,Z 618.44,A -85,B 0,C 180,E1 -13129.651,E2 -13129.651} C_VEL
LIN {X 0,Y 361.113,Z 624.562,A -85,B 0,C 180,E1 -13131.607,E2 -13131.607} C_VEL
LIN {X 0,Y 360.648,Z 629.218,A -85,B 0,C 180,E1 -13133.647,E2 -13133.647} C_VEL
LIN {X 0,Y 360.464,Z 632.121,A -85,B 0,C 180,E1 -13135.527,E2 -13135.527} C_VEL
LIN {X 0,Y 360.302,Z 633.222,A -85,B 0,C 180,E1 -13136.645,E2 -13136.645} C_VEL
LIN {X 0,Y 360.245,Z 633.902,A -85,B 0,C 180,E1 -13137.764,E2 -13137.764} C_VEL
LIN {X 0,Y 360.254,Z 634.163,A -85,B 0,C 180,E1 -13138.882,E2 -13138.882} C_VEL
LIN {X 0,Y 360.245,Z 633.944,A -85,B 0,C 180,E1 -13140,E2 -13140} C_VEL
LIN {X 0,Y 360.252,Z 633.293,A -85,B 0,C 180,E1 -13141.118,E2 -13141.118} C_VEL
LIN {X 0,Y 360.23,Z 632.22,A -85,B 0,C 180,E1 -13142.236,E2 -13142.236} C_VEL
LIN {X 0,Y 360.347,Z 629.726,A -85,B 0,C 180,E1 -13143.914,E2 -13143.914} C_VEL
LIN {X 0,Y 360.414,Z 626.14,A -85,B 0,C 180,E1 -13145.595,E2 -13145.595} C_VEL
LIN {X 0,Y 360.621,Z 621.352,A -85,B 0,C 180,E1 -13147.278,E2 -13147.278} C_VEL
LIN {X 0,Y 360.949,Z 615.231,A -85,B 0,C 180,E1 -13148.961,E2 -13148.961} C_VEL
LIN {X 0,Y 361.386,Z 607.577,A -85,B 0,C 180,E1 -13150.647,E2 -13150.647} C_VEL
LIN {X 0,Y 361.956,Z 599.749,A -85,B 0,C 180,E1 -13152.048,E2 -13152.048} C_VEL
LIN {X 0,Y 362.738,Z 589.133,A -85,B 0,C 180,E1 -13153.587,E2 -13153.587} C_VEL
LIN {X 0,Y 363.433,Z 578.998,A -85,B 0,C 180,E1 -13154.781,E2 -13154.781} C_VEL
LIN {X 0,Y 364.098,Z 568.02,A -85,B 0,C 180,E1 -13155.822,E2 -13155.822} C_VEL
LIN {X 0,Y 364.872,Z 554.938,A -85,B 0,C 180,E1 -13156.794,E2 -13156.794} C_VEL
LIN {X 0,Y 365.512,Z 541.56,A -85,B 0,C 180,E1 -13157.52,E2 -13157.52} C_VEL
LIN {X 0,Y 366.064,Z 528.791,A -85,B 0,C 180,E1 -13157.998,E2 -13157.998} C_VEL
LIN {X 0,Y 367.894,Z 445.947,A -85,B 0,C 180,E1 -13160.124,E2 -13160.124} C_VEL
LIN {X 0,Y 364.851,Z 420.66,A -85,B 0,C 180,E1 -13160.937,E2 -13160.937} C_VEL
LIN {X 0,Y 366.109,Z 399.757,A -85,B 0,C 180,E1 -13164.376,E2 -13164.376} C_VEL
LIN {X 0,Y 367.406,Z 380.498,A -85,B 0,C 180,E1 -13167.585,E2 -13167.585} C_VEL
LIN {X 0,Y 367.016,Z 376.712,A -85,B 0,C 180,E1 -13168.252,E2 -13168.252} C_VEL
LIN {X 0,Y 362.951,Z 358.903,A -85,B 0,C 180,E1 -13171.569,E2 -13171.569} C_VEL
LIN {X 0,Y 361.906,Z 354.148,A -85,B 0,C 180,E1 -13172.525,E2 -13172.525} C_VEL
LIN {X 0,Y 361.874,Z 354.034,A -85,B 0,C 180,E1 -13175.636,E2 -13175.636} C_VEL
LIN {X 0,Y 361.874,Z 354.033,A -85,B 0,C 180,E1 -13179.026,E2 -13179.026} C_VEL
LIN {X 0,Y 361.842,Z 354.031,A -85,B 0,C 180,E1 -13182.828,E2 -13182.828} C_VEL
LIN {X 0,Y 361.823,Z 354.022,A -85,B 0,C 180,E1 -13185.946,E2 -13185.946} C_VEL
LIN {X 0,Y 361.841,Z 354.028,A -85,B 0,C 180,E1 -13189.244,E2 -13189.244} C_VEL
LIN {X 0,Y 361.877,Z 354.032,A -85,B 0,C 180,E1 -13192.775,E2 -13192.775} C_VEL
LIN {X 0,Y 361.861,Z 354.037,A -85,B 0,C 180,E1 -13195.719,E2 -13195.719} C_VEL
LIN {X 0,Y 361.908,Z 354.08,A -85,B 0,C 180,E1 -13198.376,E2 -13198.376} C_VEL
LIN {X 0,Y 363.08,Z 359.016,A -85,B 0,C 180,E1 -13199.782,E2 -13199.782} C_VEL
LIN {X 0,Y 365.912,Z 371.341,A -85,B 0,C 180,E1 -13202.986,E2 -13202.986} C_VEL
LIN {X 0,Y 366.188,Z 372.596,A -85,B 0,C 180,E1 -13203.202,E2 -13203.202} C_VEL
LIN {X 0,Y 370.576,Z 383.761,A -85,B 0,C 180,E1 -13203.796,E2 -13203.796} C_VEL
LIN {X 0,Y 375,Z 406.209,A -85,B 0,C 180,E1 -13204.596,E2 -13204.596} C_VEL
LIN {X 0,Y 372.907,Z 507.969,A -85,B 0,C 180,E1 -13206.574,E2 -13206.574} C_VEL
LIN {X 0,Y 372.179,Z 522.503,A -85,B 0,C 180,E1 -13207.041,E2 -13207.041} C_VEL
LIN {X 0,Y 371.222,Z 535.757,A -85,B 0,C 180,E1 -13207.676,E2 -13207.676} C_VEL
LIN {X 0,Y 370.061,Z 549.385,A -85,B 0,C 180,E1 -13208.568,E2 -13208.568} C_VEL
LIN {X 0,Y 368.717,Z 562.154,A -85,B 0,C 180,E1 -13209.642,E2 -13209.642} C_VEL
LIN {X 0,Y 367.315,Z 573.879,A -85,B 0,C 180,E1 -13210.872,E2 -13210.872} C_VEL
LIN {X 0,Y 365.738,Z 585.58,A -85,B 0,C 180,E1 -13212.382,E2 -13212.382} C_VEL
LIN {X 0,Y 364.319,Z 596.036,A -85,B 0,C 180,E1 -13214.043,E2 -13214.043} C_VEL
LIN {X 0,Y 363.186,Z 604.661,A -85,B 0,C 180,E1 -13215.715,E2 -13215.715} C_VEL
LIN {X 0,Y 362.192,Z 612.931,A -85,B 0,C 180,E1 -13217.674,E2 -13217.674} C_VEL
LIN {X 0,Y 361.467,Z 618.697,A -85,B 0,C 180,E1 -13219.355,E2 -13219.355} C_VEL
LIN {X 0,Y 360.933,Z 623.438,A -85,B 0,C 180,E1 -13221.037,E2 -13221.037} C_VEL
LIN {X 0,Y 360.514,Z 628.345,A -85,B 0,C 180,E1 -13223.282,E2 -13223.282} C_VEL
LIN {X 0,Y 360.376,Z 631.764,A -85,B 0,C 180,E1 -13225.525,E2 -13225.525} C_VEL
LIN {X 0,Y 360.226,Z 633.799,A -85,B 0,C 180,E1 -13227.762,E2 -13227.762} C_VEL
LIN {X 0,Y 360.236,Z 634.243,A -85,B 0,C 180,E1 -13228.727,E2 -13228.727} C_VEL
LIN {X 0,Y 359.608,Z 634.54,A -85,B 0,C 180,E1 -13229.66,E2 -13229.66} C_VEL
LIN {X 0,Y 356.746,Z 634.453,A -85,B 0,C 180,E1 -13231.178,E2 -13231.178} C_VEL
LIN {X 0,Y 354.31,Z 633.864,A -85,B 0,C 180,E1 -13232.403,E2 -13232.403} C_VEL
LIN {X 0,Y 353.282,Z 633.121,A -85,B 0,C 180,E1 -13233.346,E2 -13233.346} C_VEL
LIN {X 0,Y 353.21,Z 632.81,A -85,B 0,C 180,E1 -13233.664,E2 -13233.664} C_VEL
LIN {X 0,Y 353.334,Z 630.401,A -85,B 0,C 180,E1 -13235.706,E2 -13235.706} C_VEL
LIN {X 0,Y 353.622,Z 626.315,A -85,B 0,C 180,E1 -13237.995,E2 -13237.995} C_VEL
LIN {X 0,Y 354.22,Z 620.673,A -85,B 0,C 180,E1 -13240.285,E2 -13240.285} C_VEL
LIN {X 0,Y 355.031,Z 614.31,A -85,B 0,C 180,E1 -13242.285,E2 -13242.285} C_VEL
LIN {X 0,Y 356.073,Z 606.402,A -85,B 0,C 180,E1 -13244.281,E2 -13244.281} C_VEL
LIN {X 0,Y 357.214,Z 598.122,A -85,B 0,C 180,E1 -13245.987,E2 -13245.987} C_VEL
LIN {X 0,Y 358.601,Z 588.153,A -85,B 0,C 180,E1 -13247.683,E2 -13247.683} C_VEL
LIN {X 0,Y 360.167,Z 577.057,A -85,B 0,C 180,E1 -13249.224,E2 -13249.224} C_VEL
LIN {X 0,Y 361.77,Z 564.643,A -85,B 0,C 180,E1 -13250.612,E2 -13250.612} C_VEL
LIN {X 0,Y 363.275,Z 551.501,A -85,B 0,C 180,E1 -13251.779,E2 -13251.779} C_VEL
LIN {X 0,Y 364.448,Z 538.507,A -85,B 0,C 180,E1 -13252.684,E2 -13252.684} C_VEL
LIN {X 0,Y 365.507,Z 524.703,A -85,B 0,C 180,E1 -13253.4,E2 -13253.4} C_VEL
LIN {X 0,Y 366.293,Z 511.521,A -85,B 0,C 180,E1 -13253.872,E2 -13253.872} C_VEL
LIN {X 0,Y 366.97,Z 487.298,A -85,B 0,C 180,E1 -13254.389,E2 -13254.389} C_VEL
LIN {X 0,Y 368.594,Z 407.145,A -85,B 0,C 180,E1 -13255.964,E2 -13255.964} C_VEL
LIN {X 0,Y 364.012,Z 384.745,A -85,B 0,C 180,E1 -13256.799,E2 -13256.799} C_VEL
LIN {X 0,Y 358.895,Z 372.307,A -85,B 0,C 180,E1 -13257.518,E2 -13257.518} C_VEL
LIN {X 0,Y 356.777,Z 363.021,A -85,B 0,C 180,E1 -13259.918,E2 -13259.918} C_VEL
LIN {X 0,Y 354.868,Z 355.13,A -85,B 0,C 180,E1 -13262.123,E2 -13262.123} C_VEL
LIN {X 0,Y 354.802,Z 354.911,A -85,B 0,C 180,E1 -13263.7,E2 -13263.7} C_VEL
LIN {X 0,Y 354.797,Z 354.905,A -85,B 0,C 180,E1 -13266.457,E2 -13266.457} C_VEL
LIN {X 0,Y 354.818,Z 354.897,A -85,B 0,C 180,E1 -13269.422,E2 -13269.422} C_VEL
LIN {X 0,Y 354.839,Z 354.909,A -85,B 0,C 180,E1 -13272.876,E2 -13272.876} C_VEL
LIN {X 0,Y 354.861,Z 354.885,A -85,B 0,C 180,E1 -13276.118,E2 -13276.118} C_VEL
LIN {X 0,Y 354.849,Z 354.908,A -85,B 0,C 180,E1 -13279.187,E2 -13279.187} C_VEL
LIN {X 0,Y 354.801,Z 354.878,A -85,B 0,C 180,E1 -13282.401,E2 -13282.401} C_VEL
LIN {X 0,Y 354.804,Z 354.908,A -85,B 0,C 180,E1 -13284.94,E2 -13284.94} C_VEL
LIN {X 0,Y 354.785,Z 354.904,A -85,B 0,C 180,E1 -13288.404,E2 -13288.404} C_VEL
LIN {X 0,Y 354.844,Z 354.862,A -85,B 0,C 180,E1 -13291.618,E2 -13291.618} C_VEL
LIN {X 0,Y 354.89,Z 354.895,A -85,B 0,C 180,E1 -13294.172,E2 -13294.172} C_VEL
LIN {X 0,Y 354.825,Z 354.9,A -85,B 0,C 180,E1 -13297.893,E2 -13297.893} C_VEL
LIN {X 0,Y 354.913,Z 354.898,A -85,B 0,C 180,E1 -13301.891,E2 -13301.891} C_VEL
LIN {X 0,Y 354.933,Z 354.892,A -85,B 0,C 180,E1 -13305.98,E2 -13305.98} C_VEL
LIN {X 0,Y 354.973,Z 354.876,A -85,B 0,C 180,E1 -13309.736,E2 -13309.736} C_VEL
LIN {X 0,Y 355.103,Z 354.869,A -85,B 0,C 180,E1 -13312.037,E2 -13312.037} C_VEL
LIN {X 0,Y 355.084,Z 354.876,A -85,B 0,C 180,E1 -13314.32,E2 -13314.32} C_VEL
LIN {X 0,Y 355.236,Z 354.85,A -85,B 0,C 180,E1 -13317.732,E2 -13317.732} C_VEL
LIN {X 0,Y 355.39,Z 354.839,A -85,B 0,C 180,E1 -13320,E2 -13320} C_VEL
LIN {X 0,Y 355.236,Z 354.851,A -85,B 0,C 180,E1 -13322.268,E2 -13322.268} C_VEL
LIN {X 0,Y 355.128,Z 354.874,A -85,B 0,C 180,E1 -13326.819,E2 -13326.819} C_VEL
LIN {X 0,Y 355.006,Z 354.871,A -85,B 0,C 180,E1 -13329.113,E2 -13329.113} C_VEL
LIN {X 0,Y 354.916,Z 354.898,A -85,B 0,C 180,E1 -13332.581,E2 -13332.581} C_VEL
LIN {X 0,Y 354.879,Z 354.886,A -85,B 0,C 180,E1 -13336.096,E2 -13336.096} C_VEL
LIN {X 0,Y 354.896,Z 354.901,A -85,B 0,C 180,E1 -13338.472,E2 -13338.472} C_VEL
LIN {X 0,Y 354.825,Z 354.899,A -85,B 0,C 180,E1 -13342.107,E2 -13342.107} C_VEL
LIN {X 0,Y 354.889,Z 354.895,A -85,B 0,C 180,E1 -13345.828,E2 -13345.828} C_VEL
LIN {X 0,Y 354.798,Z 354.868,A -85,B 0,C 180,E1 -13349.684,E2 -13349.684} C_VEL
LIN {X 0,Y 354.821,Z 354.911,A -85,B 0,C 180,E1 -13353.683,E2 -13353.683} C_VEL
LIN {X 0,Y 354.79,Z 354.889,A -85,B 0,C 180,E1 -13356.46,E2 -13356.46} C_VEL
LIN {X 0,Y 354.815,Z 354.893,A -85,B 0,C 180,E1 -13359.425,E2 -13359.425} C_VEL
LIN {X 0,Y 354.837,Z 354.903,A -85,B 0,C 180,E1 -13362.878,E2 -13362.878} C_VEL
LIN {X 0,Y 354.861,Z 354.891,A -85,B 0,C 180,E1 -13366.121,E2 -13366.121} C_VEL
LIN {X 0,Y 354.851,Z 354.897,A -85,B 0,C 180,E1 -13369.19,E2 -13369.19} C_VEL
LIN {X 0,Y 354.807,Z 354.915,A -85,B 0,C 180,E1 -13372.403,E2 -13372.403} C_VEL
LIN {X 0,Y 354.807,Z 354.906,A -85,B 0,C 180,E1 -13374.942,E2 -13374.942} C_VEL
LIN {X 0,Y 354.867,Z 355.027,A -85,B 0,C 180,E1 -13377.877,E2 -13377.877} C_VEL
LIN {X 0,Y 357.773,Z 367.133,A -85,B 0,C 180,E1 -13381.233,E2 -13381.233} C_VEL
LIN {X 0,Y 358.911,Z 372.302,A -85,B 0,C 180,E1 -13382.527,E2 -13382.527} C_VEL
LIN {X 0,Y 364.327,Z 385.619,A -85,B 0,C 180,E1 -13383.29,E2 -13383.29} C_VEL
LIN {X 0,Y 368.621,Z 407.616,A -85,B 0,C 180,E1 -13384.093,E2 -13384.093} C_VEL
LIN {X 0,Y 366.809,Z 492.314,A -85,B 0,C 180,E1 -13385.751,E2 -13385.751} C_VEL
LIN {X 0,Y 366.233,Z 512.434,A -85,B 0,C 180,E1 -13386.199,E2 -13386.199} C_VEL
LIN {X 0,Y 365.415,Z 526.074,A -85,B 0,C 180,E1 -13386.706,E2 -13386.706} C_VEL
LIN {X 0,Y 364.396,Z 539.07,A -85,B 0,C 180,E1 -13387.395,E2 -13387.395} C_VEL
LIN {X 0,Y 363.201,Z 551.858,A -85,B 0,C 180,E1 -13388.292,E2 -13388.292} C_VEL
LIN {X 0,Y 361.893,Z 564.183,A -85,B 0,C 180,E1 -13389.393,E2 -13389.393} C_VEL
LIN {X 0,Y 360.215,Z 576.716,A -85,B 0,C 180,E1 -13390.779,E2 -13390.779} C_VEL
LIN {X 0,Y 358.677,Z 587.881,A -85,B 0,C 180,E1 -13392.321,E2 -13392.321} C_VEL
LIN {X 0,Y 357.209,Z 597.894,A -85,B 0,C 180,E1 -13394.013,E2 -13394.013} C_VEL
LIN {X 0,Y 356.082,Z 606.235,A -85,B 0,C 180,E1 -13395.725,E2 -13395.725} C_VEL
LIN {X 0,Y 355.211,Z 613.147,A -85,B 0,C 180,E1 -13397.431,E2 -13397.431} C_VEL
LIN {X 0,Y 354.408,Z 618.886,A -85,B 0,C 180,E1 -13399.143,E2 -13399.143} C_VEL
LIN {X 0,Y 353.882,Z 623.586,A -85,B 0,C 180,E1 -13400.86,E2 -13400.86} C_VEL
LIN {X 0,Y 353.501,Z 628.46,A -85,B 0,C 180,E1 -13403.151,E2 -13403.151} C_VEL
LIN {X 0,Y 353.293,Z 631.845,A -85,B 0,C 180,E1 -13405.438,E2 -13405.438} C_VEL
LIN {X 0,Y 353.135,Z 633.842,A -85,B 0,C 180,E1 -13407.72,E2 -13407.72} C_VEL
LIN {X 0,Y 353.142,Z 634.5,A -85,B 0,C 180,E1 -13410.001,E2 -13410.001} C_VEL
LIN {X 0,Y 353.136,Z 633.83,A -85,B 0,C 180,E1 -13412.283,E2 -13412.283} C_VEL
LIN {X 0,Y 353.286,Z 631.822,A -85,B 0,C 180,E1 -13414.565,E2 -13414.565} C_VEL
LIN {X 0,Y 353.432,Z 628.429,A -85,B 0,C 180,E1 -13416.854,E2 -13416.854} C_VEL
LIN {X 0,Y 353.885,Z 623.55,A -85,B 0,C 180,E1 -13419.143,E2 -13419.143} C_VEL
LIN {X 0,Y 354.41,Z 618.839,A -85,B 0,C 180,E1 -13420.86,E2 -13420.86} C_VEL
LIN {X 0,Y 355.356,Z 612.003,A -85,B 0,C 180,E1 -13422.857,E2 -13422.857} C_VEL
LIN {X 0,Y 356.412,Z 603.519,A -85,B 0,C 180,E1 -13424.855,E2 -13424.855} C_VEL
LIN {X 0,Y 357.653,Z 594.661,A -85,B 0,C 180,E1 -13426.556,E2 -13426.556} C_VEL
LIN {X 0,Y 359.157,Z 583.931,A -85,B 0,C 180,E1 -13428.247,E2 -13428.247} C_VEL
LIN {X 0,Y 360.695,Z 573.066,A -85,B 0,C 180,E1 -13429.641,E2 -13429.641} C_VEL
LIN {X 0,Y 362.171,Z 561.284,A -85,B 0,C 180,E1 -13430.879,E2 -13430.879} C_VEL
LIN {X 0,Y 363.501,Z 548.624,A -85,B 0,C 180,E1 -13431.949,E2 -13431.949} C_VEL
LIN {X 0,Y 364.682,Z 535.292,A -85,B 0,C 180,E1 -13432.822,E2 -13432.822} C_VEL
LIN {X 0,Y 365.704,Z 520.906,A -85,B 0,C 180,E1 -13433.502,E2 -13433.502} C_VEL
LIN {X 0,Y 366.414,Z 506.784,A -85,B 0,C 180,E1 -13433.942,E2 -13433.942} C_VEL
LIN {X 0,Y 368.661,Z 408.096,A -85,B 0,C 180,E1 -13435.878,E2 -13435.878} C_VEL
LIN {X 0,Y 367.327,Z 400.374,A -85,B 0,C 180,E1 -13436.159,E2 -13436.159} C_VEL
LIN {X 0,Y 367.657,Z 390.735,A -85,B 0,C 180,E1 -13437.098,E2 -13437.098} C_VEL
LIN {X 0,Y 367.626,Z 388.907,A -85,B 0,C 180,E1 -13437.312,E2 -13437.312} C_VEL
LIN {X 0,Y 366.005,Z 382.56,A -85,B 0,C 180,E1 -13438.377,E2 -13438.377} C_VEL
LIN {X 0,Y 363.189,Z 371.359,A -85,B 0,C 180,E1 -13440.658,E2 -13440.658} C_VEL
LIN {X 0,Y 362.298,Z 368.473,A -85,B 0,C 180,E1 -13441.402,E2 -13441.402} C_VEL
LIN {X 0,Y 359.755,Z 363.81,A -85,B 0,C 180,E1 -13443.162,E2 -13443.162} C_VEL
LIN {X 0,Y 357.893,Z 360.682,A -85,B 0,C 180,E1 -13444.715,E2 -13444.715} C_VEL
LIN {X 0,Y 356.292,Z 358.452,A -85,B 0,C 180,E1 -13446.283,E2 -13446.283} C_VEL
LIN {X 0,Y 355.302,Z 356.738,A -85,B 0,C 180,E1 -13447.822,E2 -13447.822} C_VEL
LIN {X 0,Y 354.88,Z 355.186,A -85,B 0,C 180,E1 -13449.694,E2 -13449.694} C_VEL
LIN {X 0,Y 354.817,Z 355.111,A -85,B 0,C 180,E1 -13453.19,E2 -13453.19} C_VEL
LIN {X 0,Y 354.954,Z 355.877,A -85,B 0,C 180,E1 -13454.538,E2 -13454.538} C_VEL
LIN {X 0,Y 356.077,Z 358.164,A -85,B 0,C 180,E1 -13456.911,E2 -13456.911} C_VEL
LIN {X 0,Y 357.026,Z 359.333,A -85,B 0,C 180,E1 -13457.988,E2 -13457.988} C_VEL
LIN {X 0,Y 359.012,Z 363.806,A -85,B 0,C 180,E1 -13460.511,E2 -13460.511} C_VEL
LIN {X 0,Y 361.284,Z 369.355,A -85,B 0,C 180,E1 -13462.912,E2 -13462.912} C_VEL
LIN {X 0,Y 363.539,Z 375.553,A -85,B 0,C 180,E1 -13465.112,E2 -13465.112} C_VEL
LIN {X 0,Y 365.377,Z 381.879,A -85,B 0,C 180,E1 -13467.011,E2 -13467.011} C_VEL
LIN {X 0,Y 367.181,Z 390.006,A -85,B 0,C 180,E1 -13469.141,E2 -13469.141} C_VEL
LIN {X 0,Y 367.738,Z 394.635,A -85,B 0,C 180,E1 -13470.205,E2 -13470.205} C_VEL
LIN {X 0,Y 364.894,Z 415.784,A -85,B 0,C 180,E1 -13474.043,E2 -13474.043} C_VEL
LIN {X 0,Y 364.478,Z 420.126,A -85,B 0,C 180,E1 -13474.776,E2 -13474.776} C_VEL
LIN {X 0,Y 367.6,Z 435.59,A -85,B 0,C 180,E1 -13475.85,E2 -13475.85} C_VEL
LIN {X 0,Y 369.356,Z 447.906,A -85,B 0,C 180,E1 -13476.549,E2 -13476.549} C_VEL
LIN {X 0,Y 369.602,Z 451.517,A -85,B 0,C 180,E1 -13476.719,E2 -13476.719} C_VEL
LIN {X 0,Y 364.969,Z 533.369,A -85,B 0,C 180,E1 -13479.241,E2 -13479.241} C_VEL
LIN {X 0,Y 363.841,Z 547.03,A -85,B 0,C 180,E1 -13479.875,E2 -13479.875} C_VEL
LIN {X 0,Y 362.722,Z 558.741,A -85,B 0,C 180,E1 -13480.621,E2 -13480.621} C_VEL
LIN {X 0,Y 361.439,Z 570.436,A -85,B 0,C 180,E1 -13481.58,E2 -13481.58} C_VEL
